;FOLD PLACE 3
;FOLD PROPRIEDADES
Ponto_STR[Pallet_2,Prdt_32BarPacking,3].NumCaixas = 3
Ponto_STR[Pallet_2,Prdt_32BarPacking,3].PickOp = 2
Ponto_STR[Pallet_2,Prdt_32BarPacking,3].ConfGarraOp = 3
Ponto_STR[Pallet_2,Prdt_32BarPacking,3].FechaGarraOp = 0
Ponto_STR[Pallet_2,Prdt_32BarPacking,3].AbreGarraOp = 0
Ponto_STR[Pallet_2,Prdt_32BarPacking,3].SensoresCaixa = 12345
Ponto_STR[Pallet_2,Prdt_32BarPacking,3].TravaGarra = False
Ponto_STR[Pallet_2,Prdt_32BarPacking,3].SkipGoHome = False
Ponto_STR[Pallet_2,Prdt_32BarPacking,3].SkipSobeRelAtual = False
Ponto_STR[Pallet_2,Prdt_32BarPacking,3].XApp1Place=P2_32BarPacking_3_App1
Ponto_STR[Pallet_2,Prdt_32BarPacking,3].XApp2Place=P2_32BarPacking_3_App2
Ponto_STR[Pallet_2,Prdt_32BarPacking,3].XPlace=P2_32BarPacking_3_Place
;ENDFOLD
;FOLD OffsetPlace
Ponto_STR[Pallet_2,Prdt_32BarPacking,3].OffsetPlace.X=0
Ponto_STR[Pallet_2,Prdt_32BarPacking,3].OffsetPlace.Y=0
Ponto_STR[Pallet_2,Prdt_32BarPacking,3].OffsetPlace.Z=0
Ponto_STR[Pallet_2,Prdt_32BarPacking,3].OffsetPlace.A=0
Ponto_STR[Pallet_2,Prdt_32BarPacking,3].OffsetPlace.B=0
Ponto_STR[Pallet_2,Prdt_32BarPacking,3].OffsetPlace.C=0
;ENDFOLD
;ENDFOLD

;ENDFOLD
;ENDFOLD

;FOLD Pallet 2 - Produto 33BarPacking
;FOLD LAYER 1: PLACE 1 ate 2
;FOLD PLACE 1
;FOLD PROPRIEDADES
Ponto_STR[Pallet_2,Prdt_33BarPacking,1].NumCaixas = 3
Ponto_STR[Pallet_2,Prdt_33BarPacking,1].PickOp = 2
Ponto_STR[Pallet_2,Prdt_33BarPacking,1].ConfGarraOp = 2
Ponto_STR[Pallet_2,Prdt_33BarPacking,1].FechaGarraOp = 0
Ponto_STR[Pallet_2,Prdt_33BarPacking,1].AbreGarraOp = 0
Ponto_STR[Pallet_2,Prdt_33BarPacking,1].SensoresCaixa = 12345
Ponto_STR[Pallet_2,Prdt_33BarPacking,1].TravaGarra = False
Ponto_STR[Pallet_2,Prdt_33BarPacking,1].SkipGoHome = False
Ponto_STR[Pallet_2,Prdt_33BarPacking,1].SkipSobeRelAtual = False
Ponto_STR[Pallet_2,Prdt_33BarPacking,1].XApp1Place=P2_33BarPacking_1_App1
Ponto_STR[Pallet_2,Prdt_33BarPacking,1].XApp2Place=P2_33BarPacking_1_App2
Ponto_STR[Pallet_2,Prdt_33BarPacking,1].XPlace=P2_33BarPacking_1_Place
;ENDFOLD
;FOLD OffsetPlace
Ponto_STR[Pallet_2,Prdt_33BarPacking,1].OffsetPlace.X=0
Ponto_STR[Pallet_2,Prdt_33BarPacking,1].OffsetPlace.Y=0
Ponto_STR[Pallet_2,Prdt_33BarPacking,1].OffsetPlace.Z=0
Ponto_STR[Pallet_2,Prdt_33BarPacking,1].OffsetPlace.A=0
Ponto_STR[Pallet_2,Prdt_33BarPacking,1].OffsetPlace.B=0
Ponto_STR[Pallet_2,Prdt_33BarPacking,1].OffsetPlace.C=0
;ENDFOLD
;ENDFOLD

;FOLD PLACE 2
;FOLD PROPRIEDADES
Ponto_STR[Pallet_2,Prdt_33BarPacking,2].NumCaixas = 3
Ponto_STR[Pallet_2,Prdt_33BarPacking,2].PickOp = 2
Ponto_STR[Pallet_2,Prdt_33BarPacking,2].ConfGarraOp = 2
Ponto_STR[Pallet_2,Prdt_33BarPacking,2].FechaGarraOp = 0
Ponto_STR[Pallet_2,Prdt_33BarPacking,2].AbreGarraOp = 0
Ponto_STR[Pallet_2,Prdt_33BarPacking,2].SensoresCaixa = 12345
Ponto_STR[Pallet_2,Prdt_33BarPacking,2].TravaGarra = False
Ponto_STR[Pallet_2,Prdt_33BarPacking,2].SkipGoHome = False
Ponto_STR[Pallet_2,Prdt_33BarPacking,2].SkipSobeRelAtual = False
Ponto_STR[Pallet_2,Prdt_33BarPacking,2].XApp1Place=P2_33BarPacking_2_App1
Ponto_STR[Pallet_2,Prdt_33BarPacking,2].XApp2Place=P2_33BarPacking_2_App2
Ponto_STR[Pallet_2,Prdt_33BarPacking,2].XPlace=P2_33BarPacking_2_Place
;ENDFOLD
;FOLD OffsetPlace
Ponto_STR[Pallet_2,Prdt_33BarPacking,2].OffsetPlace.X=0
Ponto_STR[Pallet_2,Prdt_33BarPacking,2].OffsetPlace.Y=0
Ponto_STR[Pallet_2,Prdt_33BarPacking,2].OffsetPlace.Z=0
Ponto_STR[Pallet_2,Prdt_33BarPacking,2].OffsetPlace.A=0
Ponto_STR[Pallet_2,Prdt_33BarPacking,2].OffsetPlace.B=0
Ponto_STR[Pallet_2,Prdt_33BarPacking,2].OffsetPlace.C=0
;ENDFOLD
;ENDFOLD

;ENDFOLD
;ENDFOLD

;FOLD Pallet 2 - Produto 34BarPacking
;FOLD LAYER 1: PLACE 1 ate 2
;FOLD PLACE 1
;FOLD PROPRIEDADES
Ponto_STR[Pallet_2,Prdt_34BarPacking,1].NumCaixas = 1
Ponto_STR[Pallet_2,Prdt_34BarPacking,1].PickOp = 3
Ponto_STR[Pallet_2,Prdt_34BarPacking,1].ConfGarraOp = 3
Ponto_STR[Pallet_2,Prdt_34BarPacking,1].FechaGarraOp = 0
Ponto_STR[Pallet_2,Prdt_34BarPacking,1].AbreGarraOp = 0
Ponto_STR[Pallet_2,Prdt_34BarPacking,1].SensoresCaixa = 123
Ponto_STR[Pallet_2,Prdt_34BarPacking,1].TravaGarra = False
Ponto_STR[Pallet_2,Prdt_34BarPacking,1].SkipGoHome = False
Ponto_STR[Pallet_2,Prdt_34BarPacking,1].SkipSobeRelAtual = False
Ponto_STR[Pallet_2,Prdt_34BarPacking,1].XApp1Place=P2_34BarPacking_1_App1
Ponto_STR[Pallet_2,Prdt_34BarPacking,1].XApp2Place=P2_34BarPacking_1_App2
Ponto_STR[Pallet_2,Prdt_34BarPacking,1].XPlace=P2_34BarPacking_1_Place
;ENDFOLD
;FOLD OffsetPlace
Ponto_STR[Pallet_2,Prdt_34BarPacking,1].OffsetPlace.X=0
Ponto_STR[Pallet_2,Prdt_34BarPacking,1].OffsetPlace.Y=0
Ponto_STR[Pallet_2,Prdt_34BarPacking,1].OffsetPlace.Z=0
Ponto_STR[Pallet_2,Prdt_34BarPacking,1].OffsetPlace.A=0
Ponto_STR[Pallet_2,Prdt_34BarPacking,1].OffsetPlace.B=0
Ponto_STR[Pallet_2,Prdt_34BarPacking,1].OffsetPlace.C=0
;ENDFOLD
;ENDFOLD

;FOLD PLACE 2
;FOLD PROPRIEDADES
Ponto_STR[Pallet_2,Prdt_34BarPacking,2].NumCaixas = 1
Ponto_STR[Pallet_2,Prdt_34BarPacking,2].PickOp = 3
Ponto_STR[Pallet_2,Prdt_34BarPacking,2].ConfGarraOp = 3
Ponto_STR[Pallet_2,Prdt_34BarPacking,2].FechaGarraOp = 0
Ponto_STR[Pallet_2,Prdt_34BarPacking,2].AbreGarraOp = 0
Ponto_STR[Pallet_2,Prdt_34BarPacking,2].SensoresCaixa = 123
Ponto_STR[Pallet_2,Prdt_34BarPacking,2].TravaGarra = False
Ponto_STR[Pallet_2,Prdt_34BarPacking,2].SkipGoHome = False
Ponto_STR[Pallet_2,Prdt_34BarPacking,2].SkipSobeRelAtual = False
Ponto_STR[Pallet_2,Prdt_34BarPacking,2].XApp1Place=P2_34BarPacking_2_App1
Ponto_STR[Pallet_2,Prdt_34BarPacking,2].XApp2Place=P2_34BarPacking_2_App2
Ponto_STR[Pallet_2,Prdt_34BarPacking,2].XPlace=P2_34BarPacking_2_Place
;ENDFOLD
;FOLD OffsetPlace
Ponto_STR[Pallet_2,Prdt_34BarPacking,2].OffsetPlace.X=0
Ponto_STR[Pallet_2,Prdt_34BarPacking,2].OffsetPlace.Y=0
Ponto_STR[Pallet_2,Prdt_34BarPacking,2].OffsetPlace.Z=0
Ponto_STR[Pallet_2,Prdt_34BarPacking,2].OffsetPlace.A=0
Ponto_STR[Pallet_2,Prdt_34BarPacking,2].OffsetPlace.B=0
Ponto_STR[Pallet_2,Prdt_34BarPacking,2].OffsetPlace.C=0
;ENDFOLD
;ENDFOLD

;ENDFOLD
;ENDFOLD

;FOLD Pallet 2 - Produto 9Aero
;FOLD LAYER 1: PLACE 1 ate 2
;FOLD PLACE 1
;FOLD PROPRIEDADES
Ponto_STR[Pallet_2,Prdt_9Aero,1].NumCaixas = 4
Ponto_STR[Pallet_2,Prdt_9Aero,1].PickOp = 3
Ponto_STR[Pallet_2,Prdt_9Aero,1].ConfGarraOp = 3
Ponto_STR[Pallet_2,Prdt_9Aero,1].FechaGarraOp = 0
Ponto_STR[Pallet_2,Prdt_9Aero,1].AbreGarraOp = 0
Ponto_STR[Pallet_2,Prdt_9Aero,1].SensoresCaixa = 123456
Ponto_STR[Pallet_2,Prdt_9Aero,1].TravaGarra = False
Ponto_STR[Pallet_2,Prdt_9Aero,1].SkipGoHome = False
Ponto_STR[Pallet_2,Prdt_9Aero,1].SkipSobeRelAtual = False
Ponto_STR[Pallet_2,Prdt_9Aero,1].XApp1Place=P2_9Aero_1_App1
Ponto_STR[Pallet_2,Prdt_9Aero,1].XApp2Place=P2_9Aero_1_App2
Ponto_STR[Pallet_2,Prdt_9Aero,1].XPlace=P2_9Aero_1_Place
;ENDFOLD
;FOLD OffsetPlace
Ponto_STR[Pallet_2,Prdt_9Aero,1].OffsetPlace.X=0
Ponto_STR[Pallet_2,Prdt_9Aero,1].OffsetPlace.Y=0
Ponto_STR[Pallet_2,Prdt_9Aero,1].OffsetPlace.Z=0
Ponto_STR[Pallet_2,Prdt_9Aero,1].OffsetPlace.A=0
Ponto_STR[Pallet_2,Prdt_9Aero,1].OffsetPlace.B=0
Ponto_STR[Pallet_2,Prdt_9Aero,1].OffsetPlace.C=0
;ENDFOLD
;ENDFOLD

;FOLD PLACE 2
;FOLD PROPRIEDADES
Ponto_STR[Pallet_2,Prdt_9Aero,2].NumCaixas = 4
Ponto_STR[Pallet_2,Prdt_9Aero,2].PickOp = 3
Ponto_STR[Pallet_2,Prdt_9Aero,2].ConfGarraOp = 3
Ponto_STR[Pallet_2,Prdt_9Aero,2].FechaGarraOp = 0
Ponto_STR[Pallet_2,Prdt_9Aero,2].AbreGarraOp = 0
Ponto_STR[Pallet_2,Prdt_9Aero,2].SensoresCaixa = 123456
Ponto_STR[Pallet_2,Prdt_9Aero,2].TravaGarra = False
Ponto_STR[Pallet_2,Prdt_9Aero,2].SkipGoHome = False
Ponto_STR[Pallet_2,Prdt_9Aero,2].SkipSobeRelAtual = False
Ponto_STR[Pallet_2,Prdt_9Aero,2].XApp1Place=P2_9Aero_2_App1
Ponto_STR[Pallet_2,Prdt_9Aero,2].XApp2Place=P2_9Aero_2_App2
Ponto_STR[Pallet_2,Prdt_9Aero,2].XPlace=P2_9Aero_2_Place
;ENDFOLD
;FOLD OffsetPlace
Ponto_STR[Pallet_2,Prdt_9Aero,2].OffsetPlace.X=0
Ponto_STR[Pallet_2,Prdt_9Aero,2].OffsetPlace.Y=0
Ponto_STR[Pallet_2,Prdt_9Aero,2].OffsetPlace.Z=0
Ponto_STR[Pallet_2,Prdt_9Aero,2].OffsetPlace.A=0
Ponto_STR[Pallet_2,Prdt_9Aero,2].OffsetPlace.B=0
Ponto_STR[Pallet_2,Prdt_9Aero,2].OffsetPlace.C=0
;ENDFOLD
;ENDFOLD

;ENDFOLD
;ENDFOLD

;FOLD Pallet 2 - Produto 23Smarties
;FOLD LAYER 1: PLACE 1 ate 4
;FOLD PLACE 1
;FOLD PROPRIEDADES
Ponto_STR[Pallet_2,Prdt_23Smarties,1].NumCaixas = 2
Ponto_STR[Pallet_2,Prdt_23Smarties,1].PickOp = 4
Ponto_STR[Pallet_2,Prdt_23Smarties,1].ConfGarraOp = 4
Ponto_STR[Pallet_2,Prdt_23Smarties,1].FechaGarraOp = 0
Ponto_STR[Pallet_2,Prdt_23Smarties,1].AbreGarraOp = 0
Ponto_STR[Pallet_2,Prdt_23Smarties,1].SensoresCaixa = 456
Ponto_STR[Pallet_2,Prdt_23Smarties,1].TravaGarra = False
Ponto_STR[Pallet_2,Prdt_23Smarties,1].SkipGoHome = False
Ponto_STR[Pallet_2,Prdt_23Smarties,1].SkipSobeRelAtual = False
Ponto_STR[Pallet_2,Prdt_23Smarties,1].XApp1Place=P2_23Smarties_1_App1
Ponto_STR[Pallet_2,Prdt_23Smarties,1].XApp2Place=P2_23Smarties_1_App2
Ponto_STR[Pallet_2,Prdt_23Smarties,1].XPlace=P2_23Smarties_1_Place
;ENDFOLD
;FOLD OffsetPlace
Ponto_STR[Pallet_2,Prdt_23Smarties,1].OffsetPlace.X=0
Ponto_STR[Pallet_2,Prdt_23Smarties,1].OffsetPlace.Y=0
Ponto_STR[Pallet_2,Prdt_23Smarties,1].OffsetPlace.Z=0
Ponto_STR[Pallet_2,Prdt_23Smarties,1].OffsetPlace.A=0
Ponto_STR[Pallet_2,Prdt_23Smarties,1].OffsetPlace.B=0
Ponto_STR[Pallet_2,Prdt_23Smarties,1].OffsetPlace.C=0
;ENDFOLD
;ENDFOLD

;FOLD PLACE 2
;FOLD PROPRIEDADES
Ponto_STR[Pallet_2,Prdt_23Smarties,2].NumCaixas = 3
Ponto_STR[Pallet_2,Prdt_23Smarties,2].PickOp = 4
Ponto_STR[Pallet_2,Prdt_23Smarties,2].ConfGarraOp = 4
Ponto_STR[Pallet_2,Prdt_23Smarties,2].FechaGarraOp = 0
Ponto_STR[Pallet_2,Prdt_23Smarties,2].AbreGarraOp = 0
Ponto_STR[Pallet_2,Prdt_23Smarties,2].SensoresCaixa = 3456
Ponto_STR[Pallet_2,Prdt_23Smarties,2].TravaGarra = False
Ponto_STR[Pallet_2,Prdt_23Smarties,2].SkipGoHome = False
Ponto_STR[Pallet_2,Prdt_23Smarties,2].SkipSobeRelAtual = False
Ponto_STR[Pallet_2,Prdt_23Smarties,2].XApp1Place=P2_23Smarties_2_App1
Ponto_STR[Pallet_2,Prdt_23Smarties,2].XApp2Place=P2_23Smarties_2_App2
Ponto_STR[Pallet_2,Prdt_23Smarties,2].XPlace=P2_23Smarties_2_Place
;ENDFOLD
;FOLD OffsetPlace
Ponto_STR[Pallet_2,Prdt_23Smarties,2].OffsetPlace.X=0
Ponto_STR[Pallet_2,Prdt_23Smarties,2].OffsetPlace.Y=0
Ponto_STR[Pallet_2,Prdt_23Smarties,2].OffsetPlace.Z=0
Ponto_STR[Pallet_2,Prdt_23Smarties,2].OffsetPlace.A=0
Ponto_STR[Pallet_2,Prdt_23Smarties,2].OffsetPlace.B=0
Ponto_STR[Pallet_2,Prdt_23Smarties,2].OffsetPlace.C=0
;ENDFOLD
;ENDFOLD

;FOLD PLACE 3
;FOLD PROPRIEDADES
Ponto_STR[Pallet_2,Prdt_23Smarties,3].NumCaixas = 2
Ponto_STR[Pallet_2,Prdt_23Smarties,3].PickOp = 4
Ponto_STR[Pallet_2,Prdt_23Smarties,3].ConfGarraOp = 4
Ponto_STR[Pallet_2,Prdt_23Smarties,3].FechaGarraOp = 0
Ponto_STR[Pallet_2,Prdt_23Smarties,3].AbreGarraOp = 0
Ponto_STR[Pallet_2,Prdt_23Smarties,3].SensoresCaixa = 456
Ponto_STR[Pallet_2,Prdt_23Smarties,3].TravaGarra = False
Ponto_STR[Pallet_2,Prdt_23Smarties,3].SkipGoHome = False
Ponto_STR[Pallet_2,Prdt_23Smarties,3].SkipSobeRelAtual = False
Ponto_STR[Pallet_2,Prdt_23Smarties,3].XApp1Place=P2_23Smarties_3_App1
Ponto_STR[Pallet_2,Prdt_23Smarties,3].XApp2Place=P2_23Smarties_3_App2
Ponto_STR[Pallet_2,Prdt_23Smarties,3].XPlace=P2_23Smarties_3_Place
;ENDFOLD
;FOLD OffsetPlace
Ponto_STR[Pallet_2,Prdt_23Smarties,3].OffsetPlace.X=0
Ponto_STR[Pallet_2,Prdt_23Smarties,3].OffsetPlace.Y=0
Ponto_STR[Pallet_2,Prdt_23Smarties,3].OffsetPlace.Z=0
Ponto_STR[Pallet_2,Prdt_23Smarties,3].OffsetPlace.A=0
Ponto_STR[Pallet_2,Prdt_23Smarties,3].OffsetPlace.B=0
Ponto_STR[Pallet_2,Prdt_23Smarties,3].OffsetPlace.C=0
;ENDFOLD
;ENDFOLD

;FOLD PLACE 4
;FOLD PROPRIEDADES
Ponto_STR[Pallet_2,Prdt_23Smarties,4].NumCaixas = 3
Ponto_STR[Pallet_2,Prdt_23Smarties,4].PickOp = 4
Ponto_STR[Pallet_2,Prdt_23Smarties,4].ConfGarraOp = 4
Ponto_STR[Pallet_2,Prdt_23Smarties,4].FechaGarraOp = 0
Ponto_STR[Pallet_2,Prdt_23Smarties,4].AbreGarraOp = 0
Ponto_STR[Pallet_2,Prdt_23Smarties,4].SensoresCaixa = 3456
Ponto_STR[Pallet_2,Prdt_23Smarties,4].TravaGarra = False
Ponto_STR[Pallet_2,Prdt_23Smarties,4].SkipGoHome = False
Ponto_STR[Pallet_2,Prdt_23Smarties,4].SkipSobeRelAtual = False
Ponto_STR[Pallet_2,Prdt_23Smarties,4].XApp1Place=P2_23Smarties_4_App1
Ponto_STR[Pallet_2,Prdt_23Smarties,4].XApp2Place=P2_23Smarties_4_App2
Ponto_STR[Pallet_2,Prdt_23Smarties,4].XPlace=P2_23Smarties_4_Place
;ENDFOLD
;FOLD OffsetPlace
Ponto_STR[Pallet_2,Prdt_23Smarties,4].OffsetPlace.X=0
Ponto_STR[Pallet_2,Prdt_23Smarties,4].OffsetPlace.Y=0
Ponto_STR[Pallet_2,Prdt_23Smarties,4].OffsetPlace.Z=0
Ponto_STR[Pallet_2,Prdt_23Smarties,4].OffsetPlace.A=0
Ponto_STR[Pallet_2,Prdt_23Smarties,4].OffsetPlace.B=0
Ponto_STR[Pallet_2,Prdt_23Smarties,4].OffsetPlace.C=0
;ENDFOLD
;ENDFOLD

;ENDFOLD
;FOLD LAYER 2: PLACE 5 ate 8
;FOLD PLACE 5
;FOLD PROPRIEDADES
Ponto_STR[Pallet_2,Prdt_23Smarties,5].NumCaixas = 2
Ponto_STR[Pallet_2,Prdt_23Smarties,5].PickOp = 5
Ponto_STR[Pallet_2,Prdt_23Smarties,5].ConfGarraOp = 4
Ponto_STR[Pallet_2,Prdt_23Smarties,5].FechaGarraOp = 0
Ponto_STR[Pallet_2,Prdt_23Smarties,5].AbreGarraOp = 0
Ponto_STR[Pallet_2,Prdt_23Smarties,5].SensoresCaixa = 123
Ponto_STR[Pallet_2,Prdt_23Smarties,5].TravaGarra = False
Ponto_STR[Pallet_2,Prdt_23Smarties,5].SkipGoHome = False
Ponto_STR[Pallet_2,Prdt_23Smarties,5].SkipSobeRelAtual = False
Ponto_STR[Pallet_2,Prdt_23Smarties,5].XApp1Place=P2_23Smarties_5_App1
Ponto_STR[Pallet_2,Prdt_23Smarties,5].XApp2Place=P2_23Smarties_5_App2
Ponto_STR[Pallet_2,Prdt_23Smarties,5].XPlace=P2_23Smarties_5_Place
;ENDFOLD
;FOLD OffsetPlace
Ponto_STR[Pallet_2,Prdt_23Smarties,5].OffsetPlace.X=0
Ponto_STR[Pallet_2,Prdt_23Smarties,5].OffsetPlace.Y=0
Ponto_STR[Pallet_2,Prdt_23Smarties,5].OffsetPlace.Z=0
Ponto_STR[Pallet_2,Prdt_23Smarties,5].OffsetPlace.A=0
Ponto_STR[Pallet_2,Prdt_23Smarties,5].OffsetPlace.B=0
Ponto_STR[Pallet_2,Prdt_23Smarties,5].OffsetPlace.C=0
;ENDFOLD
;ENDFOLD

;FOLD PLACE 6
;FOLD PROPRIEDADES
Ponto_STR[Pallet_2,Prdt_23Smarties,6].NumCaixas = 3
Ponto_STR[Pallet_2,Prdt_23Smarties,6].PickOp = 5
Ponto_STR[Pallet_2,Prdt_23Smarties,6].ConfGarraOp = 4
Ponto_STR[Pallet_2,Prdt_23Smarties,6].FechaGarraOp = 0
Ponto_STR[Pallet_2,Prdt_23Smarties,6].AbreGarraOp = 0
Ponto_STR[Pallet_2,Prdt_23Smarties,6].SensoresCaixa = 1234
Ponto_STR[Pallet_2,Prdt_23Smarties,6].TravaGarra = False
Ponto_STR[Pallet_2,Prdt_23Smarties,6].SkipGoHome = False
Ponto_STR[Pallet_2,Prdt_23Smarties,6].SkipSobeRelAtual = False
Ponto_STR[Pallet_2,Prdt_23Smarties,6].XApp1Place=P2_23Smarties_6_App1
Ponto_STR[Pallet_2,Prdt_23Smarties,6].XApp2Place=P2_23Smarties_6_App2
Ponto_STR[Pallet_2,Prdt_23Smarties,6].XPlace=P2_23Smarties_6_Place
;ENDFOLD
;FOLD OffsetPlace
Ponto_STR[Pallet_2,Prdt_23Smarties,6].OffsetPlace.X=0
Ponto_STR[Pallet_2,Prdt_23Smarties,6].OffsetPlace.Y=0
Ponto_STR[Pallet_2,Prdt_23Smarties,6].OffsetPlace.Z=0
Ponto_STR[Pallet_2,Prdt_23Smarties,6].OffsetPlace.A=0
Ponto_STR[Pallet_2,Prdt_23Smarties,6].OffsetPlace.B=0
Ponto_STR[Pallet_2,Prdt_23Smarties,6].OffsetPlace.C=0
;ENDFOLD
;ENDFOLD

;FOLD PLACE 7
;FOLD PROPRIEDADES
Ponto_STR[Pallet_2,Prdt_23Smarties,7].NumCaixas = 2
Ponto_STR[Pallet_2,Prdt_23Smarties,7].PickOp = 5
Ponto_STR[Pallet_2,Prdt_23Smarties,7].ConfGarraOp = 4
Ponto_STR[Pallet_2,Prdt_23Smarties,7].FechaGarraOp = 0
Ponto_STR[Pallet_2,Prdt_23Smarties,7].AbreGarraOp = 0
Ponto_STR[Pallet_2,Prdt_23Smarties,7].SensoresCaixa = 123
Ponto_STR[Pallet_2,Prdt_23Smarties,7].TravaGarra = False
Ponto_STR[Pallet_2,Prdt_23Smarties,7].SkipGoHome = False
Ponto_STR[Pallet_2,Prdt_23Smarties,7].SkipSobeRelAtual = False
Ponto_STR[Pallet_2,Prdt_23Smarties,7].XApp1Place=P2_23Smarties_7_App1
Ponto_STR[Pallet_2,Prdt_23Smarties,7].XApp2Place=P2_23Smarties_7_App2
Ponto_STR[Pallet_2,Prdt_23Smarties,7].XPlace=P2_23Smarties_7_Place
;ENDFOLD
;FOLD OffsetPlace
Ponto_STR[Pallet_2,Prdt_23Smarties,7].OffsetPlace.X=0
Ponto_STR[Pallet_2,Prdt_23Smarties,7].OffsetPlace.Y=0
Ponto_STR[Pallet_2,Prdt_23Smarties,7].OffsetPlace.Z=0
Ponto_STR[Pallet_2,Prdt_23Smarties,7].OffsetPlace.A=0
Ponto_STR[Pallet_2,Prdt_23Smarties,7].OffsetPlace.B=0
Ponto_STR[Pallet_2,Prdt_23Smarties,7].OffsetPlace.C=0
;ENDFOLD
;ENDFOLD

;FOLD PLACE 8
;FOLD PROPRIEDADES
Ponto_STR[Pallet_2,Prdt_23Smarties,8].NumCaixas = 3
Ponto_STR[Pallet_2,Prdt_23Smarties,8].PickOp = 5
Ponto_STR[Pallet_2,Prdt_23Smarties,8].ConfGarraOp = 4
Ponto_STR[Pallet_2,Prdt_23Smarties,8].FechaGarraOp = 0
Ponto_STR[Pallet_2,Prdt_23Smarties,8].AbreGarraOp = 0
Ponto_STR[Pallet_2,Prdt_23Smarties,8].SensoresCaixa = 1234
Ponto_STR[Pallet_2,Prdt_23Smarties,8].TravaGarra = False
Ponto_STR[Pallet_2,Prdt_23Smarties,8].SkipGoHome = False
Ponto_STR[Pallet_2,Prdt_23Smarties,8].SkipSobeRelAtual = False
Ponto_STR[Pallet_2,Prdt_23Smarties,8].XApp1Place=P2_23Smarties_8_App1
Ponto_STR[Pallet_2,Prdt_23Smarties,8].XApp2Place=P2_23Smarties_8_App2
Ponto_STR[Pallet_2,Prdt_23Smarties,8].XPlace=P2_23Smarties_8_Place
;ENDFOLD
;FOLD OffsetPlace
Ponto_STR[Pallet_2,Prdt_23Smarties,8].OffsetPlace.X=0
Ponto_STR[Pallet_2,Prdt_23Smarties,8].OffsetPlace.Y=0
Ponto_STR[Pallet_2,Prdt_23Smarties,8].OffsetPlace.Z=0
Ponto_STR[Pallet_2,Prdt_23Smarties,8].OffsetPlace.A=0
Ponto_STR[Pallet_2,Prdt_23Smarties,8].OffsetPlace.B=0
Ponto_STR[Pallet_2,Prdt_23Smarties,8].OffsetPlace.C=0
;ENDFOLD
;ENDFOLD

;ENDFOLD
;ENDFOLD

;FOLD Pallet 2 - Produto 10CoffeCrisp
;FOLD LAYER 1: PLACE 1 ate 4
;FOLD PLACE 1
;FOLD PROPRIEDADES
Ponto_STR[Pallet_2,Prdt_10CoffeCrisp,1].NumCaixas = 1
Ponto_STR[Pallet_2,Prdt_10CoffeCrisp,1].PickOp = 6
Ponto_STR[Pallet_2,Prdt_10CoffeCrisp,1].ConfGarraOp = 0
Ponto_STR[Pallet_2,Prdt_10CoffeCrisp,1].FechaGarraOp = 0
Ponto_STR[Pallet_2,Prdt_10CoffeCrisp,1].AbreGarraOp = 0
Ponto_STR[Pallet_2,Prdt_10CoffeCrisp,1].SensoresCaixa = 56
Ponto_STR[Pallet_2,Prdt_10CoffeCrisp,1].TravaGarra = False
Ponto_STR[Pallet_2,Prdt_10CoffeCrisp,1].SkipGoHome = False
Ponto_STR[Pallet_2,Prdt_10CoffeCrisp,1].SkipSobeRelAtual = False
Ponto_STR[Pallet_2,Prdt_10CoffeCrisp,1].XApp1Place=P2_10CoffeCrisp_1_App1
Ponto_STR[Pallet_2,Prdt_10CoffeCrisp,1].XApp2Place=P2_10CoffeCrisp_1_App2
Ponto_STR[Pallet_2,Prdt_10CoffeCrisp,1].XPlace=P2_10CoffeCrisp_1_Place
;ENDFOLD
;FOLD OffsetPlace
Ponto_STR[Pallet_2,Prdt_10CoffeCrisp,1].OffsetPlace.X=0
Ponto_STR[Pallet_2,Prdt_10CoffeCrisp,1].OffsetPlace.Y=0
Ponto_STR[Pallet_2,Prdt_10CoffeCrisp,1].OffsetPlace.Z=0
Ponto_STR[Pallet_2,Prdt_10CoffeCrisp,1].OffsetPlace.A=0
Ponto_STR[Pallet_2,Prdt_10CoffeCrisp,1].OffsetPlace.B=0
Ponto_STR[Pallet_2,Prdt_10CoffeCrisp,1].OffsetPlace.C=0
;ENDFOLD
;ENDFOLD

;FOLD PLACE 2
;FOLD PROPRIEDADES
Ponto_STR[Pallet_2,Prdt_10CoffeCrisp,2].NumCaixas = 1
Ponto_STR[Pallet_2,Prdt_10CoffeCrisp,2].PickOp = 6
Ponto_STR[Pallet_2,Prdt_10CoffeCrisp,2].ConfGarraOp = 0
Ponto_STR[Pallet_2,Prdt_10CoffeCrisp,2].FechaGarraOp = 0
Ponto_STR[Pallet_2,Prdt_10CoffeCrisp,2].AbreGarraOp = 0
Ponto_STR[Pallet_2,Prdt_10CoffeCrisp,2].SensoresCaixa = 56
Ponto_STR[Pallet_2,Prdt_10CoffeCrisp,2].TravaGarra = False
Ponto_STR[Pallet_2,Prdt_10CoffeCrisp,2].SkipGoHome = False
Ponto_STR[Pallet_2,Prdt_10CoffeCrisp,2].SkipSobeRelAtual = False
Ponto_STR[Pallet_2,Prdt_10CoffeCrisp,2].XApp1Place=P2_10CoffeCrisp_2_App1
Ponto_STR[Pallet_2,Prdt_10CoffeCrisp,2].XApp2Place=P2_10CoffeCrisp_2_App2
Ponto_STR[Pallet_2,Prdt_10CoffeCrisp,2].XPlace=P2_10CoffeCrisp_2_Place
;ENDFOLD
;FOLD OffsetPlace
Ponto_STR[Pallet_2,Prdt_10CoffeCrisp,2].OffsetPlace.X=0
Ponto_STR[Pallet_2,Prdt_10CoffeCrisp,2].OffsetPlace.Y=0
Ponto_STR[Pallet_2,Prdt_10CoffeCrisp,2].OffsetPlace.Z=0
Ponto_STR[Pallet_2,Prdt_10CoffeCrisp,2].OffsetPlace.A=0
Ponto_STR[Pallet_2,Prdt_10CoffeCrisp,2].OffsetPlace.B=0
Ponto_STR[Pallet_2,Prdt_10CoffeCrisp,2].OffsetPlace.C=0
;ENDFOLD
;ENDFOLD

;FOLD PLACE 3
;FOLD PROPRIEDADES
Ponto_STR[Pallet_2,Prdt_10CoffeCrisp,3].NumCaixas = 3
Ponto_STR[Pallet_2,Prdt_10CoffeCrisp,3].PickOp = 1
Ponto_STR[Pallet_2,Prdt_10CoffeCrisp,3].ConfGarraOp = 0
Ponto_STR[Pallet_2,Prdt_10CoffeCrisp,3].FechaGarraOp = 0
Ponto_STR[Pallet_2,Prdt_10CoffeCrisp,3].AbreGarraOp = 0
Ponto_STR[Pallet_2,Prdt_10CoffeCrisp,3].SensoresCaixa = 12345
Ponto_STR[Pallet_2,Prdt_10CoffeCrisp,3].TravaGarra = False
Ponto_STR[Pallet_2,Prdt_10CoffeCrisp,3].SkipGoHome = False
Ponto_STR[Pallet_2,Prdt_10CoffeCrisp,3].SkipSobeRelAtual = False
Ponto_STR[Pallet_2,Prdt_10CoffeCrisp,3].XApp1Place=P2_10CoffeCrisp_3_App1
Ponto_STR[Pallet_2,Prdt_10CoffeCrisp,3].XApp2Place=P2_10CoffeCrisp_3_App2
Ponto_STR[Pallet_2,Prdt_10CoffeCrisp,3].XPlace=P2_10CoffeCrisp_3_Place
;ENDFOLD
;FOLD OffsetPlace
Ponto_STR[Pallet_2,Prdt_10CoffeCrisp,3].OffsetPlace.X=0
Ponto_STR[Pallet_2,Prdt_10CoffeCrisp,3].OffsetPlace.Y=0
Ponto_STR[Pallet_2,Prdt_10CoffeCrisp,3].OffsetPlace.Z=0
Ponto_STR[Pallet_2,Prdt_10CoffeCrisp,3].OffsetPlace.A=0
Ponto_STR[Pallet_2,Prdt_10CoffeCrisp,3].OffsetPlace.B=0
Ponto_STR[Pallet_2,Prdt_10CoffeCrisp,3].OffsetPlace.C=0
;ENDFOLD
;ENDFOLD

;FOLD PLACE 4
;FOLD PROPRIEDADES
Ponto_STR[Pallet_2,Prdt_10CoffeCrisp,4].NumCaixas = 3
Ponto_STR[Pallet_2,Prdt_10CoffeCrisp,4].PickOp = 1
Ponto_STR[Pallet_2,Prdt_10CoffeCrisp,4].ConfGarraOp = 0
Ponto_STR[Pallet_2,Prdt_10CoffeCrisp,4].FechaGarraOp = 0
Ponto_STR[Pallet_2,Prdt_10CoffeCrisp,4].AbreGarraOp = 0
Ponto_STR[Pallet_2,Prdt_10CoffeCrisp,4].SensoresCaixa = 12345
Ponto_STR[Pallet_2,Prdt_10CoffeCrisp,4].TravaGarra = False
Ponto_STR[Pallet_2,Prdt_10CoffeCrisp,4].SkipGoHome = False
Ponto_STR[Pallet_2,Prdt_10CoffeCrisp,4].SkipSobeRelAtual = False
Ponto_STR[Pallet_2,Prdt_10CoffeCrisp,4].XApp1Place=P2_10CoffeCrisp_4_App1
Ponto_STR[Pallet_2,Prdt_10CoffeCrisp,4].XApp2Place=P2_10CoffeCrisp_4_App2
Ponto_STR[Pallet_2,Prdt_10CoffeCrisp,4].XPlace=P2_10CoffeCrisp_4_Place
;ENDFOLD
;FOLD OffsetPlace
Ponto_STR[Pallet_2,Prdt_10CoffeCrisp,4].OffsetPlace.X=0
Ponto_STR[Pallet_2,Prdt_10CoffeCrisp,4].OffsetPlace.Y=0
Ponto_STR[Pallet_2,Prdt_10CoffeCrisp,4].OffsetPlace.Z=0
Ponto_STR[Pallet_2,Prdt_10CoffeCrisp,4].OffsetPlace.A=0
Ponto_STR[Pallet_2,Prdt_10CoffeCrisp,4].OffsetPlace.B=0
Ponto_STR[Pallet_2,Prdt_10CoffeCrisp,4].OffsetPlace.C=0
;ENDFOLD
;ENDFOLD

;ENDFOLD
;FOLD LAYER 2: PLACE 5 ate 8
;FOLD PLACE 5
;FOLD PROPRIEDADES
Ponto_STR[Pallet_2,Prdt_10CoffeCrisp,5].NumCaixas = 1
Ponto_STR[Pallet_2,Prdt_10CoffeCrisp,5].PickOp = 3
Ponto_STR[Pallet_2,Prdt_10CoffeCrisp,5].ConfGarraOp = 3
Ponto_STR[Pallet_2,Prdt_10CoffeCrisp,5].FechaGarraOp = 0
Ponto_STR[Pallet_2,Prdt_10CoffeCrisp,5].AbreGarraOp = 0
Ponto_STR[Pallet_2,Prdt_10CoffeCrisp,5].SensoresCaixa = 12
Ponto_STR[Pallet_2,Prdt_10CoffeCrisp,5].TravaGarra = False
Ponto_STR[Pallet_2,Prdt_10CoffeCrisp,5].SkipGoHome = False
Ponto_STR[Pallet_2,Prdt_10CoffeCrisp,5].SkipSobeRelAtual = False
Ponto_STR[Pallet_2,Prdt_10CoffeCrisp,5].XApp1Place=P2_10CoffeCrisp_5_App1
Ponto_STR[Pallet_2,Prdt_10CoffeCrisp,5].XApp2Place=P2_10CoffeCrisp_5_App2
Ponto_STR[Pallet_2,Prdt_10CoffeCrisp,5].XPlace=P2_10CoffeCrisp_5_Place
;ENDFOLD
;FOLD OffsetPlace
Ponto_STR[Pallet_2,Prdt_10CoffeCrisp,5].OffsetPlace.X=0
Ponto_STR[Pallet_2,Prdt_10CoffeCrisp,5].OffsetPlace.Y=0
Ponto_STR[Pallet_2,Prdt_10CoffeCrisp,5].OffsetPlace.Z=0
Ponto_STR[Pallet_2,Prdt_10CoffeCrisp,5].OffsetPlace.A=0
Ponto_STR[Pallet_2,Prdt_10CoffeCrisp,5].OffsetPlace.B=0
Ponto_STR[Pallet_2,Prdt_10CoffeCrisp,5].OffsetPlace.C=0
;ENDFOLD
;ENDFOLD

;FOLD PLACE 6
;FOLD PROPRIEDADES
Ponto_STR[Pallet_2,Prdt_10CoffeCrisp,6].NumCaixas = 1
Ponto_STR[Pallet_2,Prdt_10CoffeCrisp,6].PickOp = 3
Ponto_STR[Pallet_2,Prdt_10CoffeCrisp,6].ConfGarraOp = 3
Ponto_STR[Pallet_2,Prdt_10CoffeCrisp,6].FechaGarraOp = 0
Ponto_STR[Pallet_2,Prdt_10CoffeCrisp,6].AbreGarraOp = 0
Ponto_STR[Pallet_2,Prdt_10CoffeCrisp,6].SensoresCaixa = 12
Ponto_STR[Pallet_2,Prdt_10CoffeCrisp,6].TravaGarra = False
Ponto_STR[Pallet_2,Prdt_10CoffeCrisp,6].SkipGoHome = False
Ponto_STR[Pallet_2,Prdt_10CoffeCrisp,6].SkipSobeRelAtual = False
Ponto_STR[Pallet_2,Prdt_10CoffeCrisp,6].XApp1Place=P2_10CoffeCrisp_6_App1
Ponto_STR[Pallet_2,Prdt_10CoffeCrisp,6].XApp2Place=P2_10CoffeCrisp_6_App2
Ponto_STR[Pallet_2,Prdt_10CoffeCrisp,6].XPlace=P2_10CoffeCrisp_6_Place
;ENDFOLD
;FOLD OffsetPlace
Ponto_STR[Pallet_2,Prdt_10CoffeCrisp,6].OffsetPlace.X=0
Ponto_STR[Pallet_2,Prdt_10CoffeCrisp,6].OffsetPlace.Y=0
Ponto_STR[Pallet_2,Prdt_10CoffeCrisp,6].OffsetPlace.Z=0
Ponto_STR[Pallet_2,Prdt_10CoffeCrisp,6].OffsetPlace.A=0
Ponto_STR[Pallet_2,Prdt_10CoffeCrisp,6].OffsetPlace.B=0
Ponto_STR[Pallet_2,Prdt_10CoffeCrisp,6].OffsetPlace.C=0
;ENDFOLD
;ENDFOLD

;FOLD PLACE 7
;FOLD PROPRIEDADES
Ponto_STR[Pallet_2,Prdt_10CoffeCrisp,7].NumCaixas = 3
Ponto_STR[Pallet_2,Prdt_10CoffeCrisp,7].PickOp = 1
Ponto_STR[Pallet_2,Prdt_10CoffeCrisp,7].ConfGarraOp = 0
Ponto_STR[Pallet_2,Prdt_10CoffeCrisp,7].FechaGarraOp = 0
Ponto_STR[Pallet_2,Prdt_10CoffeCrisp,7].AbreGarraOp = 1
Ponto_STR[Pallet_2,Prdt_10CoffeCrisp,7].SensoresCaixa = 12345
Ponto_STR[Pallet_2,Prdt_10CoffeCrisp,7].TravaGarra = True
Ponto_STR[Pallet_2,Prdt_10CoffeCrisp,7].SkipGoHome = False
Ponto_STR[Pallet_2,Prdt_10CoffeCrisp,7].SkipSobeRelAtual = False
Ponto_STR[Pallet_2,Prdt_10CoffeCrisp,7].XApp1Place=P2_10CoffeCrisp_7_App1
Ponto_STR[Pallet_2,Prdt_10CoffeCrisp,7].XApp2Place=P2_10CoffeCrisp_7_App2
Ponto_STR[Pallet_2,Prdt_10CoffeCrisp,7].XPlace=P2_10CoffeCrisp_7_Place
;ENDFOLD
;FOLD OffsetPlace
Ponto_STR[Pallet_2,Prdt_10CoffeCrisp,7].OffsetPlace.X=0
Ponto_STR[Pallet_2,Prdt_10CoffeCrisp,7].OffsetPlace.Y=0
Ponto_STR[Pallet_2,Prdt_10CoffeCrisp,7].OffsetPlace.Z=0
Ponto_STR[Pallet_2,Prdt_10CoffeCrisp,7].OffsetPlace.A=0
Ponto_STR[Pallet_2,Prdt_10CoffeCrisp,7].OffsetPlace.B=0
Ponto_STR[Pallet_2,Prdt_10CoffeCrisp,7].OffsetPlace.C=0
;ENDFOLD
;ENDFOLD

;FOLD PLACE 8
;FOLD PROPRIEDADES
Ponto_STR[Pallet_2,Prdt_10CoffeCrisp,8].NumCaixas = 3
Ponto_STR[Pallet_2,Prdt_10CoffeCrisp,8].PickOp = 1
Ponto_STR[Pallet_2,Prdt_10CoffeCrisp,8].ConfGarraOp = 0
Ponto_STR[Pallet_2,Prdt_10CoffeCrisp,8].FechaGarraOp = 0
Ponto_STR[Pallet_2,Prdt_10CoffeCrisp,8].AbreGarraOp = 1
Ponto_STR[Pallet_2,Prdt_10CoffeCrisp,8].SensoresCaixa = 12345
Ponto_STR[Pallet_2,Prdt_10CoffeCrisp,8].TravaGarra = True
Ponto_STR[Pallet_2,Prdt_10CoffeCrisp,8].SkipGoHome = False
Ponto_STR[Pallet_2,Prdt_10CoffeCrisp,8].SkipSobeRelAtual = False
Ponto_STR[Pallet_2,Prdt_10CoffeCrisp,8].XApp1Place=P2_10CoffeCrisp_8_App1
Ponto_STR[Pallet_2,Prdt_10CoffeCrisp,8].XApp2Place=P2_10CoffeCrisp_8_App2
Ponto_STR[Pallet_2,Prdt_10CoffeCrisp,8].XPlace=P2_10CoffeCrisp_8_Place
;ENDFOLD
;FOLD OffsetPlace
Ponto_STR[Pallet_2,Prdt_10CoffeCrisp,8].OffsetPlace.X=0
Ponto_STR[Pallet_2,Prdt_10CoffeCrisp,8].OffsetPlace.Y=0
Ponto_STR[Pallet_2,Prdt_10CoffeCrisp,8].OffsetPlace.Z=0
Ponto_STR[Pallet_2,Prdt_10CoffeCrisp,8].OffsetPlace.A=0
Ponto_STR[Pallet_2,Prdt_10CoffeCrisp,8].OffsetPlace.B=0
Ponto_STR[Pallet_2,Prdt_10CoffeCrisp,8].OffsetPlace.C=0
;ENDFOLD
;ENDFOLD

;ENDFOLD
;ENDFOLD

;FOLD Pallet 2 - Produto 19KitKat
;FOLD LAYER 1: PLACE 1 ate 6
;FOLD PLACE 1
;FOLD PROPRIEDADES
Ponto_STR[Pallet_2,Prdt_19KitKat,1].NumCaixas = 1
Ponto_STR[Pallet_2,Prdt_19KitKat,1].PickOp = 6
Ponto_STR[Pallet_2,Prdt_19KitKat,1].ConfGarraOp = 0
Ponto_STR[Pallet_2,Prdt_19KitKat,1].FechaGarraOp = 0
Ponto_STR[Pallet_2,Prdt_19KitKat,1].AbreGarraOp = 0
Ponto_STR[Pallet_2,Prdt_19KitKat,1].SensoresCaixa = 6
Ponto_STR[Pallet_2,Prdt_19KitKat,1].TravaGarra = False
Ponto_STR[Pallet_2,Prdt_19KitKat,1].SkipGoHome = False
Ponto_STR[Pallet_2,Prdt_19KitKat,1].SkipSobeRelAtual = False
Ponto_STR[Pallet_2,Prdt_19KitKat,1].XApp1Place=P2_19KitKat_1_App1
Ponto_STR[Pallet_2,Prdt_19KitKat,1].XApp2Place=P2_19KitKat_1_App2
Ponto_STR[Pallet_2,Prdt_19KitKat,1].XPlace=P2_19KitKat_1_Place
;ENDFOLD
;FOLD OffsetPlace
Ponto_STR[Pallet_2,Prdt_19KitKat,1].OffsetPlace.X=0
Ponto_STR[Pallet_2,Prdt_19KitKat,1].OffsetPlace.Y=0
Ponto_STR[Pallet_2,Prdt_19KitKat,1].OffsetPlace.Z=0
Ponto_STR[Pallet_2,Prdt_19KitKat,1].OffsetPlace.A=0
Ponto_STR[Pallet_2,Prdt_19KitKat,1].OffsetPlace.B=0
Ponto_STR[Pallet_2,Prdt_19KitKat,1].OffsetPlace.C=0
;ENDFOLD
;ENDFOLD

;FOLD PLACE 2
;FOLD PROPRIEDADES
Ponto_STR[Pallet_2,Prdt_19KitKat,2].NumCaixas = 1
Ponto_STR[Pallet_2,Prdt_19KitKat,2].PickOp = 6
Ponto_STR[Pallet_2,Prdt_19KitKat,2].ConfGarraOp = 0
Ponto_STR[Pallet_2,Prdt_19KitKat,2].FechaGarraOp = 0
Ponto_STR[Pallet_2,Prdt_19KitKat,2].AbreGarraOp = 0
Ponto_STR[Pallet_2,Prdt_19KitKat,2].SensoresCaixa = 6
Ponto_STR[Pallet_2,Prdt_19KitKat,2].TravaGarra = False
Ponto_STR[Pallet_2,Prdt_19KitKat,2].SkipGoHome = False
Ponto_STR[Pallet_2,Prdt_19KitKat,2].SkipSobeRelAtual = False
Ponto_STR[Pallet_2,Prdt_19KitKat,2].XApp1Place=P2_19KitKat_2_App1
Ponto_STR[Pallet_2,Prdt_19KitKat,2].XApp2Place=P2_19KitKat_2_App2
Ponto_STR[Pallet_2,Prdt_19KitKat,2].XPlace=P2_19KitKat_2_Place
;ENDFOLD
;FOLD OffsetPlace
Ponto_STR[Pallet_2,Prdt_19KitKat,2].OffsetPlace.X=0
Ponto_STR[Pallet_2,Prdt_19KitKat,2].OffsetPlace.Y=0
Ponto_STR[Pallet_2,Prdt_19KitKat,2].OffsetPlace.Z=0
Ponto_STR[Pallet_2,Prdt_19KitKat,2].OffsetPlace.A=0
Ponto_STR[Pallet_2,Prdt_19KitKat,2].OffsetPlace.B=0
Ponto_STR[Pallet_2,Prdt_19KitKat,2].OffsetPlace.C=0
;ENDFOLD
;ENDFOLD

;FOLD PLACE 3
;FOLD PROPRIEDADES
Ponto_STR[Pallet_2,Prdt_19KitKat,3].NumCaixas = 1
Ponto_STR[Pallet_2,Prdt_19KitKat,3].PickOp = 6
Ponto_STR[Pallet_2,Prdt_19KitKat,3].ConfGarraOp = 0
Ponto_STR[Pallet_2,Prdt_19KitKat,3].FechaGarraOp = 0
Ponto_STR[Pallet_2,Prdt_19KitKat,3].AbreGarraOp = 0
Ponto_STR[Pallet_2,Prdt_19KitKat,3].SensoresCaixa = 6
Ponto_STR[Pallet_2,Prdt_19KitKat,3].TravaGarra = False
Ponto_STR[Pallet_2,Prdt_19KitKat,3].SkipGoHome = False
Ponto_STR[Pallet_2,Prdt_19KitKat,3].SkipSobeRelAtual = False
Ponto_STR[Pallet_2,Prdt_19KitKat,3].XApp1Place=P2_19KitKat_3_App1
Ponto_STR[Pallet_2,Prdt_19KitKat,3].XApp2Place=P2_19KitKat_3_App2
Ponto_STR[Pallet_2,Prdt_19KitKat,3].XPlace=P2_19KitKat_3_Place
;ENDFOLD
;FOLD OffsetPlace
Ponto_STR[Pallet_2,Prdt_19KitKat,3].OffsetPlace.X=0
Ponto_STR[Pallet_2,Prdt_19KitKat,3].OffsetPlace.Y=0
Ponto_STR[Pallet_2,Prdt_19KitKat,3].OffsetPlace.Z=0
Ponto_STR[Pallet_2,Prdt_19KitKat,3].OffsetPlace.A=0
Ponto_STR[Pallet_2,Prdt_19KitKat,3].OffsetPlace.B=0
Ponto_STR[Pallet_2,Prdt_19KitKat,3].OffsetPlace.C=0
;ENDFOLD
;ENDFOLD

;FOLD PLACE 4
;FOLD PROPRIEDADES
Ponto_STR[Pallet_2,Prdt_19KitKat,4].NumCaixas = 4
Ponto_STR[Pallet_2,Prdt_19KitKat,4].PickOp = 1
Ponto_STR[Pallet_2,Prdt_19KitKat,4].ConfGarraOp = 0
Ponto_STR[Pallet_2,Prdt_19KitKat,4].FechaGarraOp = 0
Ponto_STR[Pallet_2,Prdt_19KitKat,4].AbreGarraOp = 0
Ponto_STR[Pallet_2,Prdt_19KitKat,4].SensoresCaixa = 12345
Ponto_STR[Pallet_2,Prdt_19KitKat,4].TravaGarra = False
Ponto_STR[Pallet_2,Prdt_19KitKat,4].SkipGoHome = False
Ponto_STR[Pallet_2,Prdt_19KitKat,4].SkipSobeRelAtual = False
Ponto_STR[Pallet_2,Prdt_19KitKat,4].XApp1Place=P2_19KitKat_4_App1
Ponto_STR[Pallet_2,Prdt_19KitKat,4].XApp2Place=P2_19KitKat_4_App2
Ponto_STR[Pallet_2,Prdt_19KitKat,4].XPlace=P2_19KitKat_4_Place
;ENDFOLD
;FOLD OffsetPlace
Ponto_STR[Pallet_2,Prdt_19KitKat,4].OffsetPlace.X=0
Ponto_STR[Pallet_2,Prdt_19KitKat,4].OffsetPlace.Y=0
Ponto_STR[Pallet_2,Prdt_19KitKat,4].OffsetPlace.Z=0
Ponto_STR[Pallet_2,Prdt_19KitKat,4].OffsetPlace.A=0
Ponto_STR[Pallet_2,Prdt_19KitKat,4].OffsetPlace.B=0
Ponto_STR[Pallet_2,Prdt_19KitKat,4].OffsetPlace.C=0
;ENDFOLD
;ENDFOLD

;FOLD PLACE 5
;FOLD PROPRIEDADES
Ponto_STR[Pallet_2,Prdt_19KitKat,5].NumCaixas = 4
Ponto_STR[Pallet_2,Prdt_19KitKat,5].PickOp = 1
Ponto_STR[Pallet_2,Prdt_19KitKat,5].ConfGarraOp = 0
Ponto_STR[Pallet_2,Prdt_19KitKat,5].FechaGarraOp = 0
Ponto_STR[Pallet_2,Prdt_19KitKat,5].AbreGarraOp = 0
Ponto_STR[Pallet_2,Prdt_19KitKat,5].SensoresCaixa = 12345
Ponto_STR[Pallet_2,Prdt_19KitKat,5].TravaGarra = False
Ponto_STR[Pallet_2,Prdt_19KitKat,5].SkipGoHome = False
Ponto_STR[Pallet_2,Prdt_19KitKat,5].SkipSobeRelAtual = False
Ponto_STR[Pallet_2,Prdt_19KitKat,5].XApp1Place=P2_19KitKat_5_App1
Ponto_STR[Pallet_2,Prdt_19KitKat,5].XApp2Place=P2_19KitKat_5_App2
Ponto_STR[Pallet_2,Prdt_19KitKat,5].XPlace=P2_19KitKat_5_Place
;ENDFOLD
;FOLD OffsetPlace
Ponto_STR[Pallet_2,Prdt_19KitKat,5].OffsetPlace.X=0
Ponto_STR[Pallet_2,Prdt_19KitKat,5].OffsetPlace.Y=0
Ponto_STR[Pallet_2,Prdt_19KitKat,5].OffsetPlace.Z=0
Ponto_STR[Pallet_2,Prdt_19KitKat,5].OffsetPlace.A=0
Ponto_STR[Pallet_2,Prdt_19KitKat,5].OffsetPlace.B=0
Ponto_STR[Pallet_2,Prdt_19KitKat,5].OffsetPlace.C=0
;ENDFOLD
;ENDFOLD

;FOLD PLACE 6
;FOLD PROPRIEDADES
Ponto_STR[Pallet_2,Prdt_19KitKat,6].NumCaixas = 4
Ponto_STR[Pallet_2,Prdt_19KitKat,6].PickOp = 1
Ponto_STR[Pallet_2,Prdt_19KitKat,6].ConfGarraOp = 0
Ponto_STR[Pallet_2,Prdt_19KitKat,6].FechaGarraOp = 0
Ponto_STR[Pallet_2,Prdt_19KitKat,6].AbreGarraOp = 0
Ponto_STR[Pallet_2,Prdt_19KitKat,6].SensoresCaixa = 12345
Ponto_STR[Pallet_2,Prdt_19KitKat,6].TravaGarra = False
Ponto_STR[Pallet_2,Prdt_19KitKat,6].SkipGoHome = False
Ponto_STR[Pallet_2,Prdt_19KitKat,6].SkipSobeRelAtual = False
Ponto_STR[Pallet_2,Prdt_19KitKat,6].XApp1Place=P2_19KitKat_6_App1
Ponto_STR[Pallet_2,Prdt_19KitKat,6].XApp2Place=P2_19KitKat_6_App2
Ponto_STR[Pallet_2,Prdt_19KitKat,6].XPlace=P2_19KitKat_6_Place
;ENDFOLD
;FOLD OffsetPlace
Ponto_STR[Pallet_2,Prdt_19KitKat,6].OffsetPlace.X=0
Ponto_STR[Pallet_2,Prdt_19KitKat,6].OffsetPlace.Y=0
Ponto_STR[Pallet_2,Prdt_19KitKat,6].OffsetPlace.Z=0
Ponto_STR[Pallet_2,Prdt_19KitKat,6].OffsetPlace.A=0
Ponto_STR[Pallet_2,Prdt_19KitKat,6].OffsetPlace.B=0
Ponto_STR[Pallet_2,Prdt_19KitKat,6].OffsetPlace.C=0
;ENDFOLD
;ENDFOLD

;ENDFOLD
;FOLD LAYER 2: PLACE 7 ate 12
;FOLD PLACE 7
;FOLD PROPRIEDADES
Ponto_STR[Pallet_2,Prdt_19KitKat,7].NumCaixas = 1
Ponto_STR[Pallet_2,Prdt_19KitKat,7].PickOp = 1
Ponto_STR[Pallet_2,Prdt_19KitKat,7].ConfGarraOp = 0
Ponto_STR[Pallet_2,Prdt_19KitKat,7].FechaGarraOp = 0
Ponto_STR[Pallet_2,Prdt_19KitKat,7].AbreGarraOp = 0
Ponto_STR[Pallet_2,Prdt_19KitKat,7].SensoresCaixa = 1
Ponto_STR[Pallet_2,Prdt_19KitKat,7].TravaGarra = False
Ponto_STR[Pallet_2,Prdt_19KitKat,7].SkipGoHome = False
Ponto_STR[Pallet_2,Prdt_19KitKat,7].SkipSobeRelAtual = False
Ponto_STR[Pallet_2,Prdt_19KitKat,7].XApp1Place=P2_19KitKat_7_App1
Ponto_STR[Pallet_2,Prdt_19KitKat,7].XApp2Place=P2_19KitKat_7_App2
Ponto_STR[Pallet_2,Prdt_19KitKat,7].XPlace=P2_19KitKat_7_Place
;ENDFOLD
;FOLD OffsetPlace
Ponto_STR[Pallet_2,Prdt_19KitKat,7].OffsetPlace.X=0
Ponto_STR[Pallet_2,Prdt_19KitKat,7].OffsetPlace.Y=0
Ponto_STR[Pallet_2,Prdt_19KitKat,7].OffsetPlace.Z=0
Ponto_STR[Pallet_2,Prdt_19KitKat,7].OffsetPlace.A=0
Ponto_STR[Pallet_2,Prdt_19KitKat,7].OffsetPlace.B=0
Ponto_STR[Pallet_2,Prdt_19KitKat,7].OffsetPlace.C=0
;ENDFOLD
;ENDFOLD

;FOLD PLACE 8
;FOLD PROPRIEDADES
Ponto_STR[Pallet_2,Prdt_19KitKat,8].NumCaixas = 1
Ponto_STR[Pallet_2,Prdt_19KitKat,8].PickOp = 1
Ponto_STR[Pallet_2,Prdt_19KitKat,8].ConfGarraOp = 0
Ponto_STR[Pallet_2,Prdt_19KitKat,8].FechaGarraOp = 0
Ponto_STR[Pallet_2,Prdt_19KitKat,8].AbreGarraOp = 0
Ponto_STR[Pallet_2,Prdt_19KitKat,8].SensoresCaixa = 1
Ponto_STR[Pallet_2,Prdt_19KitKat,8].TravaGarra = False
Ponto_STR[Pallet_2,Prdt_19KitKat,8].SkipGoHome = False
Ponto_STR[Pallet_2,Prdt_19KitKat,8].SkipSobeRelAtual = False
Ponto_STR[Pallet_2,Prdt_19KitKat,8].XApp1Place=P2_19KitKat_8_App1
Ponto_STR[Pallet_2,Prdt_19KitKat,8].XApp2Place=P2_19KitKat_8_App2
Ponto_STR[Pallet_2,Prdt_19KitKat,8].XPlace=P2_19KitKat_8_Place
;ENDFOLD
;FOLD OffsetPlace
Ponto_STR[Pallet_2,Prdt_19KitKat,8].OffsetPlace.X=0
Ponto_STR[Pallet_2,Prdt_19KitKat,8].OffsetPlace.Y=0
Ponto_STR[Pallet_2,Prdt_19KitKat,8].OffsetPlace.Z=0
Ponto_STR[Pallet_2,Prdt_19KitKat,8].OffsetPlace.A=0
Ponto_STR[Pallet_2,Prdt_19KitKat,8].OffsetPlace.B=0
Ponto_STR[Pallet_2,Prdt_19KitKat,8].OffsetPlace.C=0
;ENDFOLD
;ENDFOLD

;FOLD PLACE 9
;FOLD PROPRIEDADES
Ponto_STR[Pallet_2,Prdt_19KitKat,9].NumCaixas = 1
Ponto_STR[Pallet_2,Prdt_19KitKat,9].PickOp = 1
Ponto_STR[Pallet_2,Prdt_19KitKat,9].ConfGarraOp = 0
Ponto_STR[Pallet_2,Prdt_19KitKat,9].FechaGarraOp = 0
Ponto_STR[Pallet_2,Prdt_19KitKat,9].AbreGarraOp = 0
Ponto_STR[Pallet_2,Prdt_19KitKat,9].SensoresCaixa = 1
Ponto_STR[Pallet_2,Prdt_19KitKat,9].TravaGarra = False
Ponto_STR[Pallet_2,Prdt_19KitKat,9].SkipGoHome = False
Ponto_STR[Pallet_2,Prdt_19KitKat,9].SkipSobeRelAtual = False
Ponto_STR[Pallet_2,Prdt_19KitKat,9].XApp1Place=P2_19KitKat_9_App1
Ponto_STR[Pallet_2,Prdt_19KitKat,9].XApp2Place=P2_19KitKat_9_App2
Ponto_STR[Pallet_2,Prdt_19KitKat,9].XPlace=P2_19KitKat_9_Place
;ENDFOLD
;FOLD OffsetPlace
Ponto_STR[Pallet_2,Prdt_19KitKat,9].OffsetPlace.X=0
Ponto_STR[Pallet_2,Prdt_19KitKat,9].OffsetPlace.Y=0
Ponto_STR[Pallet_2,Prdt_19KitKat,9].OffsetPlace.Z=0
Ponto_STR[Pallet_2,Prdt_19KitKat,9].OffsetPlace.A=0
Ponto_STR[Pallet_2,Prdt_19KitKat,9].OffsetPlace.B=0
Ponto_STR[Pallet_2,Prdt_19KitKat,9].OffsetPlace.C=0
;ENDFOLD
;ENDFOLD

;FOLD PLACE 10
;FOLD PROPRIEDADES
Ponto_STR[Pallet_2,Prdt_19KitKat,10].NumCaixas = 4
Ponto_STR[Pallet_2,Prdt_19KitKat,10].PickOp = 1
Ponto_STR[Pallet_2,Prdt_19KitKat,10].ConfGarraOp = 0
Ponto_STR[Pallet_2,Prdt_19KitKat,10].FechaGarraOp = 0
Ponto_STR[Pallet_2,Prdt_19KitKat,10].AbreGarraOp = 1
Ponto_STR[Pallet_2,Prdt_19KitKat,10].SensoresCaixa = 12345
Ponto_STR[Pallet_2,Prdt_19KitKat,10].TravaGarra = True
Ponto_STR[Pallet_2,Prdt_19KitKat,10].SkipGoHome = False
Ponto_STR[Pallet_2,Prdt_19KitKat,10].SkipSobeRelAtual = False
Ponto_STR[Pallet_2,Prdt_19KitKat,10].XApp1Place=P2_19KitKat_10_App1
Ponto_STR[Pallet_2,Prdt_19KitKat,10].XApp2Place=P2_19KitKat_10_App2
Ponto_STR[Pallet_2,Prdt_19KitKat,10].XPlace=P2_19KitKat_10_Place
;ENDFOLD
;FOLD OffsetPlace
Ponto_STR[Pallet_2,Prdt_19KitKat,10].OffsetPlace.X=0
Ponto_STR[Pallet_2,Prdt_19KitKat,10].OffsetPlace.Y=0
Ponto_STR[Pallet_2,Prdt_19KitKat,10].OffsetPlace.Z=0
Ponto_STR[Pallet_2,Prdt_19KitKat,10].OffsetPlace.A=0
Ponto_STR[Pallet_2,Prdt_19KitKat,10].OffsetPlace.B=0
Ponto_STR[Pallet_2,Prdt_19KitKat,10].OffsetPlace.C=0
;ENDFOLD
;ENDFOLD

;FOLD PLACE 11
;FOLD PROPRIEDADES
Ponto_STR[Pallet_2,Prdt_19KitKat,11].NumCaixas = 4
Ponto_STR[Pallet_2,Prdt_19KitKat,11].PickOp = 1
Ponto_STR[Pallet_2,Prdt_19KitKat,11].ConfGarraOp = 0
Ponto_STR[Pallet_2,Prdt_19KitKat,11].FechaGarraOp = 0
Ponto_STR[Pallet_2,Prdt_19KitKat,11].AbreGarraOp = 1
Ponto_STR[Pallet_2,Prdt_19KitKat,11].SensoresCaixa = 12345
Ponto_STR[Pallet_2,Prdt_19KitKat,11].TravaGarra = True
Ponto_STR[Pallet_2,Prdt_19KitKat,11].SkipGoHome = False
Ponto_STR[Pallet_2,Prdt_19KitKat,11].SkipSobeRelAtual = False
Ponto_STR[Pallet_2,Prdt_19KitKat,11].XApp1Place=P2_19KitKat_11_App1
Ponto_STR[Pallet_2,Prdt_19KitKat,11].XApp2Place=P2_19KitKat_11_App2
Ponto_STR[Pallet_2,Prdt_19KitKat,11].XPlace=P2_19KitKat_11_Place
;ENDFOLD
;FOLD OffsetPlace
Ponto_STR[Pallet_2,Prdt_19KitKat,11].OffsetPlace.X=0
Ponto_STR[Pallet_2,Prdt_19KitKat,11].OffsetPlace.Y=0
Ponto_STR[Pallet_2,Prdt_19KitKat,11].OffsetPlace.Z=0
Ponto_STR[Pallet_2,Prdt_19KitKat,11].OffsetPlace.A=0
Ponto_STR[Pallet_2,Prdt_19KitKat,11].OffsetPlace.B=0
Ponto_STR[Pallet_2,Prdt_19KitKat,11].OffsetPlace.C=0
;ENDFOLD
;ENDFOLD

;FOLD PLACE 12
;FOLD PROPRIEDADES
Ponto_STR[Pallet_2,Prdt_19KitKat,12].NumCaixas = 4
Ponto_STR[Pallet_2,Prdt_19KitKat,12].PickOp = 1
Ponto_STR[Pallet_2,Prdt_19KitKat,12].ConfGarraOp = 0
Ponto_STR[Pallet_2,Prdt_19KitKat,12].FechaGarraOp = 0
Ponto_STR[Pallet_2,Prdt_19KitKat,12].AbreGarraOp = 1
Ponto_STR[Pallet_2,Prdt_19KitKat,12].SensoresCaixa = 12345
Ponto_STR[Pallet_2,Prdt_19KitKat,12].TravaGarra = True
Ponto_STR[Pallet_2,Prdt_19KitKat,12].SkipGoHome = False
Ponto_STR[Pallet_2,Prdt_19KitKat,12].SkipSobeRelAtual = False
Ponto_STR[Pallet_2,Prdt_19KitKat,12].XApp1Place=P2_19KitKat_12_App1
Ponto_STR[Pallet_2,Prdt_19KitKat,12].XApp2Place=P2_19KitKat_12_App2
Ponto_STR[Pallet_2,Prdt_19KitKat,12].XPlace=P2_19KitKat_12_Place
;ENDFOLD
;FOLD OffsetPlace
Ponto_STR[Pallet_2,Prdt_19KitKat,12].OffsetPlace.X=0
Ponto_STR[Pallet_2,Prdt_19KitKat,12].OffsetPlace.Y=0
Ponto_STR[Pallet_2,Prdt_19KitKat,12].OffsetPlace.Z=0
Ponto_STR[Pallet_2,Prdt_19KitKat,12].OffsetPlace.A=0
Ponto_STR[Pallet_2,Prdt_19KitKat,12].OffsetPlace.B=0
Ponto_STR[Pallet_2,Prdt_19KitKat,12].OffsetPlace.C=0
;ENDFOLD
;ENDFOLD

;ENDFOLD
;ENDFOLD

;FOLD Pallet 2 - Produto 7Aero
;FOLD LAYER 1: PLACE 1 ate 8
;FOLD PLACE 1
;FOLD PROPRIEDADES
Ponto_STR[Pallet_2,Prdt_7Aero,1].NumCaixas = 3
Ponto_STR[Pallet_2,Prdt_7Aero,1].PickOp = 6
Ponto_STR[Pallet_2,Prdt_7Aero,1].ConfGarraOp = 0
Ponto_STR[Pallet_2,Prdt_7Aero,1].FechaGarraOp = 0
Ponto_STR[Pallet_2,Prdt_7Aero,1].AbreGarraOp = 0
Ponto_STR[Pallet_2,Prdt_7Aero,1].SensoresCaixa = 564
Ponto_STR[Pallet_2,Prdt_7Aero,1].TravaGarra = False
Ponto_STR[Pallet_2,Prdt_7Aero,1].SkipGoHome = False
Ponto_STR[Pallet_2,Prdt_7Aero,1].SkipSobeRelAtual = False
Ponto_STR[Pallet_2,Prdt_7Aero,1].XApp1Place=P2_7Aero_1_App1
Ponto_STR[Pallet_2,Prdt_7Aero,1].XApp2Place=P2_7Aero_1_App2
Ponto_STR[Pallet_2,Prdt_7Aero,1].XPlace=P2_7Aero_1_Place
;ENDFOLD
;FOLD OffsetPlace
Ponto_STR[Pallet_2,Prdt_7Aero,1].OffsetPlace.X=0
Ponto_STR[Pallet_2,Prdt_7Aero,1].OffsetPlace.Y=0
Ponto_STR[Pallet_2,Prdt_7Aero,1].OffsetPlace.Z=0
Ponto_STR[Pallet_2,Prdt_7Aero,1].OffsetPlace.A=0
Ponto_STR[Pallet_2,Prdt_7Aero,1].OffsetPlace.B=0
Ponto_STR[Pallet_2,Prdt_7Aero,1].OffsetPlace.C=0
;ENDFOLD
;ENDFOLD

;FOLD PLACE 2
;FOLD PROPRIEDADES
Ponto_STR[Pallet_2,Prdt_7Aero,2].NumCaixas = 3
Ponto_STR[Pallet_2,Prdt_7Aero,2].PickOp = 6
Ponto_STR[Pallet_2,Prdt_7Aero,2].ConfGarraOp = 0
Ponto_STR[Pallet_2,Prdt_7Aero,2].FechaGarraOp = 0
Ponto_STR[Pallet_2,Prdt_7Aero,2].AbreGarraOp = 0
Ponto_STR[Pallet_2,Prdt_7Aero,2].SensoresCaixa = 564
Ponto_STR[Pallet_2,Prdt_7Aero,2].TravaGarra = False
Ponto_STR[Pallet_2,Prdt_7Aero,2].SkipGoHome = False
Ponto_STR[Pallet_2,Prdt_7Aero,2].SkipSobeRelAtual = False
Ponto_STR[Pallet_2,Prdt_7Aero,2].XApp1Place=P2_7Aero_2_App1
Ponto_STR[Pallet_2,Prdt_7Aero,2].XApp2Place=P2_7Aero_2_App2
Ponto_STR[Pallet_2,Prdt_7Aero,2].XPlace=P2_7Aero_2_Place
;ENDFOLD
;FOLD OffsetPlace
Ponto_STR[Pallet_2,Prdt_7Aero,2].OffsetPlace.X=0
Ponto_STR[Pallet_2,Prdt_7Aero,2].OffsetPlace.Y=0
Ponto_STR[Pallet_2,Prdt_7Aero,2].OffsetPlace.Z=0
Ponto_STR[Pallet_2,Prdt_7Aero,2].OffsetPlace.A=0
Ponto_STR[Pallet_2,Prdt_7Aero,2].OffsetPlace.B=0
Ponto_STR[Pallet_2,Prdt_7Aero,2].OffsetPlace.C=0
;ENDFOLD
;ENDFOLD

;FOLD PLACE 3
;FOLD PROPRIEDADES
Ponto_STR[Pallet_2,Prdt_7Aero,3].NumCaixas = 2
Ponto_STR[Pallet_2,Prdt_7Aero,3].PickOp = 8
Ponto_STR[Pallet_2,Prdt_7Aero,3].ConfGarraOp = 5
Ponto_STR[Pallet_2,Prdt_7Aero,3].FechaGarraOp = 0
Ponto_STR[Pallet_2,Prdt_7Aero,3].AbreGarraOp = 0
Ponto_STR[Pallet_2,Prdt_7Aero,3].SensoresCaixa = 12
Ponto_STR[Pallet_2,Prdt_7Aero,3].TravaGarra = False
Ponto_STR[Pallet_2,Prdt_7Aero,3].SkipGoHome = False
Ponto_STR[Pallet_2,Prdt_7Aero,3].SkipSobeRelAtual = False
Ponto_STR[Pallet_2,Prdt_7Aero,3].XApp1Place=P2_7Aero_3_App1
Ponto_STR[Pallet_2,Prdt_7Aero,3].XApp2Place=P2_7Aero_3_App2
Ponto_STR[Pallet_2,Prdt_7Aero,3].XPlace=P2_7Aero_3_Place
;ENDFOLD
;FOLD OffsetPlace
Ponto_STR[Pallet_2,Prdt_7Aero,3].OffsetPlace.X=0
Ponto_STR[Pallet_2,Prdt_7Aero,3].OffsetPlace.Y=0
Ponto_STR[Pallet_2,Prdt_7Aero,3].OffsetPlace.Z=0
Ponto_STR[Pallet_2,Prdt_7Aero,3].OffsetPlace.A=0
Ponto_STR[Pallet_2,Prdt_7Aero,3].OffsetPlace.B=0
Ponto_STR[Pallet_2,Prdt_7Aero,3].OffsetPlace.C=0
;ENDFOLD
;ENDFOLD

;FOLD PLACE 4
;FOLD PROPRIEDADES
Ponto_STR[Pallet_2,Prdt_7Aero,4].NumCaixas = 2
Ponto_STR[Pallet_2,Prdt_7Aero,4].PickOp = 8
Ponto_STR[Pallet_2,Prdt_7Aero,4].ConfGarraOp = 5
Ponto_STR[Pallet_2,Prdt_7Aero,4].FechaGarraOp = 0
Ponto_STR[Pallet_2,Prdt_7Aero,4].AbreGarraOp = 0
Ponto_STR[Pallet_2,Prdt_7Aero,4].SensoresCaixa = 12
Ponto_STR[Pallet_2,Prdt_7Aero,4].TravaGarra = False
Ponto_STR[Pallet_2,Prdt_7Aero,4].SkipGoHome = False
Ponto_STR[Pallet_2,Prdt_7Aero,4].SkipSobeRelAtual = False
Ponto_STR[Pallet_2,Prdt_7Aero,4].XApp1Place=P2_7Aero_4_App1
Ponto_STR[Pallet_2,Prdt_7Aero,4].XApp2Place=P2_7Aero_4_App2
Ponto_STR[Pallet_2,Prdt_7Aero,4].XPlace=P2_7Aero_4_Place
;ENDFOLD
;FOLD OffsetPlace
Ponto_STR[Pallet_2,Prdt_7Aero,4].OffsetPlace.X=0
Ponto_STR[Pallet_2,Prdt_7Aero,4].OffsetPlace.Y=0
Ponto_STR[Pallet_2,Prdt_7Aero,4].OffsetPlace.Z=0
Ponto_STR[Pallet_2,Prdt_7Aero,4].OffsetPlace.A=0
Ponto_STR[Pallet_2,Prdt_7Aero,4].OffsetPlace.B=0
Ponto_STR[Pallet_2,Prdt_7Aero,4].OffsetPlace.C=0
;ENDFOLD
;ENDFOLD

;FOLD PLACE 5
;FOLD PROPRIEDADES
Ponto_STR[Pallet_2,Prdt_7Aero,5].NumCaixas = 3
Ponto_STR[Pallet_2,Prdt_7Aero,5].PickOp = 8
Ponto_STR[Pallet_2,Prdt_7Aero,5].ConfGarraOp = 5
Ponto_STR[Pallet_2,Prdt_7Aero,5].FechaGarraOp = 0
Ponto_STR[Pallet_2,Prdt_7Aero,5].AbreGarraOp = 1
Ponto_STR[Pallet_2,Prdt_7Aero,5].SensoresCaixa = 123
Ponto_STR[Pallet_2,Prdt_7Aero,5].TravaGarra = True
Ponto_STR[Pallet_2,Prdt_7Aero,5].SkipGoHome = False
Ponto_STR[Pallet_2,Prdt_7Aero,5].SkipSobeRelAtual = False
Ponto_STR[Pallet_2,Prdt_7Aero,5].XApp1Place=P2_7Aero_5_App1
Ponto_STR[Pallet_2,Prdt_7Aero,5].XApp2Place=P2_7Aero_5_App2
Ponto_STR[Pallet_2,Prdt_7Aero,5].XPlace=P2_7Aero_5_Place
;ENDFOLD
;FOLD OffsetPlace
Ponto_STR[Pallet_2,Prdt_7Aero,5].OffsetPlace.X=0
Ponto_STR[Pallet_2,Prdt_7Aero,5].OffsetPlace.Y=0
Ponto_STR[Pallet_2,Prdt_7Aero,5].OffsetPlace.Z=0
Ponto_STR[Pallet_2,Prdt_7Aero,5].OffsetPlace.A=0
Ponto_STR[Pallet_2,Prdt_7Aero,5].OffsetPlace.B=0
Ponto_STR[Pallet_2,Prdt_7Aero,5].OffsetPlace.C=0
;ENDFOLD
;ENDFOLD

;FOLD PLACE 6
;FOLD PROPRIEDADES
Ponto_STR[Pallet_2,Prdt_7Aero,6].NumCaixas = 3
Ponto_STR[Pallet_2,Prdt_7Aero,6].PickOp = 8
Ponto_STR[Pallet_2,Prdt_7Aero,6].ConfGarraOp = 5
Ponto_STR[Pallet_2,Prdt_7Aero,6].FechaGarraOp = 0
Ponto_STR[Pallet_2,Prdt_7Aero,6].AbreGarraOp = 1
Ponto_STR[Pallet_2,Prdt_7Aero,6].SensoresCaixa = 123
Ponto_STR[Pallet_2,Prdt_7Aero,6].TravaGarra = True
Ponto_STR[Pallet_2,Prdt_7Aero,6].SkipGoHome = False
Ponto_STR[Pallet_2,Prdt_7Aero,6].SkipSobeRelAtual = False
Ponto_STR[Pallet_2,Prdt_7Aero,6].XApp1Place=P2_7Aero_6_App1
Ponto_STR[Pallet_2,Prdt_7Aero,6].XApp2Place=P2_7Aero_6_App2
Ponto_STR[Pallet_2,Prdt_7Aero,6].XPlace=P2_7Aero_6_Place
;ENDFOLD
;FOLD OffsetPlace
Ponto_STR[Pallet_2,Prdt_7Aero,6].OffsetPlace.X=0
Ponto_STR[Pallet_2,Prdt_7Aero,6].OffsetPlace.Y=0
Ponto_STR[Pallet_2,Prdt_7Aero,6].OffsetPlace.Z=0
Ponto_STR[Pallet_2,Prdt_7Aero,6].OffsetPlace.A=0
Ponto_STR[Pallet_2,Prdt_7Aero,6].OffsetPlace.B=0
Ponto_STR[Pallet_2,Prdt_7Aero,6].OffsetPlace.C=0
;ENDFOLD
;ENDFOLD

;FOLD PLACE 7
;FOLD PROPRIEDADES
Ponto_STR[Pallet_2,Prdt_7Aero,7].NumCaixas = 2
Ponto_STR[Pallet_2,Prdt_7Aero,7].PickOp = 8
Ponto_STR[Pallet_2,Prdt_7Aero,7].ConfGarraOp = 5
Ponto_STR[Pallet_2,Prdt_7Aero,7].FechaGarraOp = 0
Ponto_STR[Pallet_2,Prdt_7Aero,7].AbreGarraOp = 1
Ponto_STR[Pallet_2,Prdt_7Aero,7].SensoresCaixa = 12
Ponto_STR[Pallet_2,Prdt_7Aero,7].TravaGarra = True
Ponto_STR[Pallet_2,Prdt_7Aero,7].SkipGoHome = False
Ponto_STR[Pallet_2,Prdt_7Aero,7].SkipSobeRelAtual = False
Ponto_STR[Pallet_2,Prdt_7Aero,7].XApp1Place=P2_7Aero_7_App1
Ponto_STR[Pallet_2,Prdt_7Aero,7].XApp2Place=P2_7Aero_7_App2
Ponto_STR[Pallet_2,Prdt_7Aero,7].XPlace=P2_7Aero_7_Place
;ENDFOLD
;FOLD OffsetPlace
Ponto_STR[Pallet_2,Prdt_7Aero,7].OffsetPlace.X=0
Ponto_STR[Pallet_2,Prdt_7Aero,7].OffsetPlace.Y=0
Ponto_STR[Pallet_2,Prdt_7Aero,7].OffsetPlace.Z=0
Ponto_STR[Pallet_2,Prdt_7Aero,7].OffsetPlace.A=0
Ponto_STR[Pallet_2,Prdt_7Aero,7].OffsetPlace.B=0
Ponto_STR[Pallet_2,Prdt_7Aero,7].OffsetPlace.C=0
;ENDFOLD
;ENDFOLD

;FOLD PLACE 8
;FOLD PROPRIEDADES
Ponto_STR[Pallet_2,Prdt_7Aero,8].NumCaixas = 2
Ponto_STR[Pallet_2,Prdt_7Aero,8].PickOp = 8
Ponto_STR[Pallet_2,Prdt_7Aero,8].ConfGarraOp = 5
Ponto_STR[Pallet_2,Prdt_7Aero,8].FechaGarraOp = 0
Ponto_STR[Pallet_2,Prdt_7Aero,8].AbreGarraOp = 1
Ponto_STR[Pallet_2,Prdt_7Aero,8].SensoresCaixa = 12
Ponto_STR[Pallet_2,Prdt_7Aero,8].TravaGarra = True
Ponto_STR[Pallet_2,Prdt_7Aero,8].SkipGoHome = False
Ponto_STR[Pallet_2,Prdt_7Aero,8].SkipSobeRelAtual = False
Ponto_STR[Pallet_2,Prdt_7Aero,8].XApp1Place=P2_7Aero_8_App1
Ponto_STR[Pallet_2,Prdt_7Aero,8].XApp2Place=P2_7Aero_8_App2
Ponto_STR[Pallet_2,Prdt_7Aero,8].XPlace=P2_7Aero_8_Place
;ENDFOLD
;FOLD OffsetPlace
Ponto_STR[Pallet_2,Prdt_7Aero,8].OffsetPlace.X=0
Ponto_STR[Pallet_2,Prdt_7Aero,8].OffsetPlace.Y=0
Ponto_STR[Pallet_2,Prdt_7Aero,8].OffsetPlace.Z=0
Ponto_STR[Pallet_2,Prdt_7Aero,8].OffsetPlace.A=0
Ponto_STR[Pallet_2,Prdt_7Aero,8].OffsetPlace.B=0
Ponto_STR[Pallet_2,Prdt_7Aero,8].OffsetPlace.C=0
;ENDFOLD
;ENDFOLD

;ENDFOLD
;FOLD LAYER 2: PLACE 9 ate 16
;FOLD PLACE 9
;FOLD PROPRIEDADES
Ponto_STR[Pallet_2,Prdt_7Aero,9].NumCaixas = 2
Ponto_STR[Pallet_2,Prdt_7Aero,9].PickOp = 8
Ponto_STR[Pallet_2,Prdt_7Aero,9].ConfGarraOp = 5
Ponto_STR[Pallet_2,Prdt_7Aero,9].FechaGarraOp = 0
Ponto_STR[Pallet_2,Prdt_7Aero,9].AbreGarraOp = 1
Ponto_STR[Pallet_2,Prdt_7Aero,9].SensoresCaixa = 12
Ponto_STR[Pallet_2,Prdt_7Aero,9].TravaGarra = True
Ponto_STR[Pallet_2,Prdt_7Aero,9].SkipGoHome = False
Ponto_STR[Pallet_2,Prdt_7Aero,9].SkipSobeRelAtual = False
Ponto_STR[Pallet_2,Prdt_7Aero,9].XApp1Place=P2_7Aero_9_App1
Ponto_STR[Pallet_2,Prdt_7Aero,9].XApp2Place=P2_7Aero_9_App2
Ponto_STR[Pallet_2,Prdt_7Aero,9].XPlace=P2_7Aero_9_Place
;ENDFOLD
;FOLD OffsetPlace
Ponto_STR[Pallet_2,Prdt_7Aero,9].OffsetPlace.X=0
Ponto_STR[Pallet_2,Prdt_7Aero,9].OffsetPlace.Y=0
Ponto_STR[Pallet_2,Prdt_7Aero,9].OffsetPlace.Z=0
Ponto_STR[Pallet_2,Prdt_7Aero,9].OffsetPlace.A=0
Ponto_STR[Pallet_2,Prdt_7Aero,9].OffsetPlace.B=0
Ponto_STR[Pallet_2,Prdt_7Aero,9].OffsetPlace.C=0
;ENDFOLD
;ENDFOLD

;FOLD PLACE 10
;FOLD PROPRIEDADES
Ponto_STR[Pallet_2,Prdt_7Aero,10].NumCaixas = 2
Ponto_STR[Pallet_2,Prdt_7Aero,10].PickOp = 8
Ponto_STR[Pallet_2,Prdt_7Aero,10].ConfGarraOp = 5
Ponto_STR[Pallet_2,Prdt_7Aero,10].FechaGarraOp = 0
Ponto_STR[Pallet_2,Prdt_7Aero,10].AbreGarraOp = 1
Ponto_STR[Pallet_2,Prdt_7Aero,10].SensoresCaixa = 12
Ponto_STR[Pallet_2,Prdt_7Aero,10].TravaGarra = True
Ponto_STR[Pallet_2,Prdt_7Aero,10].SkipGoHome = False
Ponto_STR[Pallet_2,Prdt_7Aero,10].SkipSobeRelAtual = False
Ponto_STR[Pallet_2,Prdt_7Aero,10].XApp1Place=P2_7Aero_10_App1
Ponto_STR[Pallet_2,Prdt_7Aero,10].XApp2Place=P2_7Aero_10_App2
Ponto_STR[Pallet_2,Prdt_7Aero,10].XPlace=P2_7Aero_10_Place
;ENDFOLD
;FOLD OffsetPlace
Ponto_STR[Pallet_2,Prdt_7Aero,10].OffsetPlace.X=0
Ponto_STR[Pallet_2,Prdt_7Aero,10].OffsetPlace.Y=0
Ponto_STR[Pallet_2,Prdt_7Aero,10].OffsetPlace.Z=0
Ponto_STR[Pallet_2,Prdt_7Aero,10].OffsetPlace.A=0
Ponto_STR[Pallet_2,Prdt_7Aero,10].OffsetPlace.B=0
Ponto_STR[Pallet_2,Prdt_7Aero,10].OffsetPlace.C=0
;ENDFOLD
;ENDFOLD

;FOLD PLACE 11
;FOLD PROPRIEDADES
Ponto_STR[Pallet_2,Prdt_7Aero,11].NumCaixas = 3
Ponto_STR[Pallet_2,Prdt_7Aero,11].PickOp = 8
Ponto_STR[Pallet_2,Prdt_7Aero,11].ConfGarraOp = 5
Ponto_STR[Pallet_2,Prdt_7Aero,11].FechaGarraOp = 0
Ponto_STR[Pallet_2,Prdt_7Aero,11].AbreGarraOp = 0
Ponto_STR[Pallet_2,Prdt_7Aero,11].SensoresCaixa = 123
Ponto_STR[Pallet_2,Prdt_7Aero,11].TravaGarra = False
Ponto_STR[Pallet_2,Prdt_7Aero,11].SkipGoHome = False
Ponto_STR[Pallet_2,Prdt_7Aero,11].SkipSobeRelAtual = False
Ponto_STR[Pallet_2,Prdt_7Aero,11].XApp1Place=P2_7Aero_11_App1
Ponto_STR[Pallet_2,Prdt_7Aero,11].XApp2Place=P2_7Aero_11_App2
Ponto_STR[Pallet_2,Prdt_7Aero,11].XPlace=P2_7Aero_11_Place
;ENDFOLD
;FOLD OffsetPlace
Ponto_STR[Pallet_2,Prdt_7Aero,11].OffsetPlace.X=0
Ponto_STR[Pallet_2,Prdt_7Aero,11].OffsetPlace.Y=0
Ponto_STR[Pallet_2,Prdt_7Aero,11].OffsetPlace.Z=0
Ponto_STR[Pallet_2,Prdt_7Aero,11].OffsetPlace.A=0
Ponto_STR[Pallet_2,Prdt_7Aero,11].OffsetPlace.B=0
Ponto_STR[Pallet_2,Prdt_7Aero,11].OffsetPlace.C=0
;ENDFOLD
;ENDFOLD

;FOLD PLACE 12
;FOLD PROPRIEDADES
Ponto_STR[Pallet_2,Prdt_7Aero,12].NumCaixas = 3
Ponto_STR[Pallet_2,Prdt_7Aero,12].PickOp = 8
Ponto_STR[Pallet_2,Prdt_7Aero,12].ConfGarraOp = 5
Ponto_STR[Pallet_2,Prdt_7Aero,12].FechaGarraOp = 0
Ponto_STR[Pallet_2,Prdt_7Aero,12].AbreGarraOp = 0
Ponto_STR[Pallet_2,Prdt_7Aero,12].SensoresCaixa = 123
Ponto_STR[Pallet_2,Prdt_7Aero,12].TravaGarra = False
Ponto_STR[Pallet_2,Prdt_7Aero,12].SkipGoHome = False
Ponto_STR[Pallet_2,Prdt_7Aero,12].SkipSobeRelAtual = False
Ponto_STR[Pallet_2,Prdt_7Aero,12].XApp1Place=P2_7Aero_12_App1
Ponto_STR[Pallet_2,Prdt_7Aero,12].XApp2Place=P2_7Aero_12_App2
Ponto_STR[Pallet_2,Prdt_7Aero,12].XPlace=P2_7Aero_12_Place
;ENDFOLD
;FOLD OffsetPlace
Ponto_STR[Pallet_2,Prdt_7Aero,12].OffsetPlace.X=0
Ponto_STR[Pallet_2,Prdt_7Aero,12].OffsetPlace.Y=0
Ponto_STR[Pallet_2,Prdt_7Aero,12].OffsetPlace.Z=0
Ponto_STR[Pallet_2,Prdt_7Aero,12].OffsetPlace.A=0
Ponto_STR[Pallet_2,Prdt_7Aero,12].OffsetPlace.B=0
Ponto_STR[Pallet_2,Prdt_7Aero,12].OffsetPlace.C=0
;ENDFOLD
;ENDFOLD

;FOLD PLACE 13
;FOLD PROPRIEDADES
Ponto_STR[Pallet_2,Prdt_7Aero,13].NumCaixas = 3
Ponto_STR[Pallet_2,Prdt_7Aero,13].PickOp = 8
Ponto_STR[Pallet_2,Prdt_7Aero,13].ConfGarraOp = 5
Ponto_STR[Pallet_2,Prdt_7Aero,13].FechaGarraOp = 0
Ponto_STR[Pallet_2,Prdt_7Aero,13].AbreGarraOp = 0
Ponto_STR[Pallet_2,Prdt_7Aero,13].SensoresCaixa = 123
Ponto_STR[Pallet_2,Prdt_7Aero,13].TravaGarra = False
Ponto_STR[Pallet_2,Prdt_7Aero,13].SkipGoHome = False
Ponto_STR[Pallet_2,Prdt_7Aero,13].SkipSobeRelAtual = False
Ponto_STR[Pallet_2,Prdt_7Aero,13].XApp1Place=P2_7Aero_13_App1
Ponto_STR[Pallet_2,Prdt_7Aero,13].XApp2Place=P2_7Aero_13_App2
Ponto_STR[Pallet_2,Prdt_7Aero,13].XPlace=P2_7Aero_13_Place
;ENDFOLD
;FOLD OffsetPlace
Ponto_STR[Pallet_2,Prdt_7Aero,13].OffsetPlace.X=0
Ponto_STR[Pallet_2,Prdt_7Aero,13].OffsetPlace.Y=0
Ponto_STR[Pallet_2,Prdt_7Aero,13].OffsetPlace.Z=0
Ponto_STR[Pallet_2,Prdt_7Aero,13].OffsetPlace.A=0
Ponto_STR[Pallet_2,Prdt_7Aero,13].OffsetPlace.B=0
Ponto_STR[Pallet_2,Prdt_7Aero,13].OffsetPlace.C=0
;ENDFOLD
;ENDFOLD

;FOLD PLACE 14
;FOLD PROPRIEDADES
Ponto_STR[Pallet_2,Prdt_7Aero,14].NumCaixas = 3
Ponto_STR[Pallet_2,Prdt_7Aero,14].PickOp = 8
Ponto_STR[Pallet_2,Prdt_7Aero,14].ConfGarraOp = 5
Ponto_STR[Pallet_2,Prdt_7Aero,14].FechaGarraOp = 0
Ponto_STR[Pallet_2,Prdt_7Aero,14].AbreGarraOp = 0
Ponto_STR[Pallet_2,Prdt_7Aero,14].SensoresCaixa = 123
Ponto_STR[Pallet_2,Prdt_7Aero,14].TravaGarra = False
Ponto_STR[Pallet_2,Prdt_7Aero,14].SkipGoHome = False
Ponto_STR[Pallet_2,Prdt_7Aero,14].SkipSobeRelAtual = False
Ponto_STR[Pallet_2,Prdt_7Aero,14].XApp1Place=P2_7Aero_14_App1
Ponto_STR[Pallet_2,Prdt_7Aero,14].XApp2Place=P2_7Aero_14_App2
Ponto_STR[Pallet_2,Prdt_7Aero,14].XPlace=P2_7Aero_14_Place
;ENDFOLD
;FOLD OffsetPlace
Ponto_STR[Pallet_2,Prdt_7Aero,14].OffsetPlace.X=0
Ponto_STR[Pallet_2,Prdt_7Aero,14].OffsetPlace.Y=0
Ponto_STR[Pallet_2,Prdt_7Aero,14].OffsetPlace.Z=0
Ponto_STR[Pallet_2,Prdt_7Aero,14].OffsetPlace.A=0
Ponto_STR[Pallet_2,Prdt_7Aero,14].OffsetPlace.B=0
Ponto_STR[Pallet_2,Prdt_7Aero,14].OffsetPlace.C=0
;ENDFOLD
;ENDFOLD

;FOLD PLACE 15
;FOLD PROPRIEDADES
Ponto_STR[Pallet_2,Prdt_7Aero,15].NumCaixas = 2
Ponto_STR[Pallet_2,Prdt_7Aero,15].PickOp = 8
Ponto_STR[Pallet_2,Prdt_7Aero,15].ConfGarraOp = 5
Ponto_STR[Pallet_2,Prdt_7Aero,15].FechaGarraOp = 0
Ponto_STR[Pallet_2,Prdt_7Aero,15].AbreGarraOp = 1
Ponto_STR[Pallet_2,Prdt_7Aero,15].SensoresCaixa = 12
Ponto_STR[Pallet_2,Prdt_7Aero,15].TravaGarra = True
Ponto_STR[Pallet_2,Prdt_7Aero,15].SkipGoHome = False
Ponto_STR[Pallet_2,Prdt_7Aero,15].SkipSobeRelAtual = False
Ponto_STR[Pallet_2,Prdt_7Aero,15].XApp1Place=P2_7Aero_15_App1
Ponto_STR[Pallet_2,Prdt_7Aero,15].XApp2Place=P2_7Aero_15_App2
Ponto_STR[Pallet_2,Prdt_7Aero,15].XPlace=P2_7Aero_15_Place
;ENDFOLD
;FOLD OffsetPlace
Ponto_STR[Pallet_2,Prdt_7Aero,15].OffsetPlace.X=0
Ponto_STR[Pallet_2,Prdt_7Aero,15].OffsetPlace.Y=0
Ponto_STR[Pallet_2,Prdt_7Aero,15].OffsetPlace.Z=0
Ponto_STR[Pallet_2,Prdt_7Aero,15].OffsetPlace.A=0
Ponto_STR[Pallet_2,Prdt_7Aero,15].OffsetPlace.B=0
Ponto_STR[Pallet_2,Prdt_7Aero,15].OffsetPlace.C=0
;ENDFOLD
;ENDFOLD

;FOLD PLACE 16
;FOLD PROPRIEDADES
Ponto_STR[Pallet_2,Prdt_7Aero,16].NumCaixas = 2
Ponto_STR[Pallet_2,Prdt_7Aero,16].PickOp = 8
Ponto_STR[Pallet_2,Prdt_7Aero,16].ConfGarraOp = 5
Ponto_STR[Pallet_2,Prdt_7Aero,16].FechaGarraOp = 0
Ponto_STR[Pallet_2,Prdt_7Aero,16].AbreGarraOp = 1
Ponto_STR[Pallet_2,Prdt_7Aero,16].SensoresCaixa = 12
Ponto_STR[Pallet_2,Prdt_7Aero,16].TravaGarra = True
Ponto_STR[Pallet_2,Prdt_7Aero,16].SkipGoHome = False
Ponto_STR[Pallet_2,Prdt_7Aero,16].SkipSobeRelAtual = False
Ponto_STR[Pallet_2,Prdt_7Aero,16].XApp1Place=P2_7Aero_16_App1
Ponto_STR[Pallet_2,Prdt_7Aero,16].XApp2Place=P2_7Aero_16_App2
Ponto_STR[Pallet_2,Prdt_7Aero,16].XPlace=P2_7Aero_16_Place
;ENDFOLD
;FOLD OffsetPlace
Ponto_STR[Pallet_2,Prdt_7Aero,16].OffsetPlace.X=0
Ponto_STR[Pallet_2,Prdt_7Aero,16].OffsetPlace.Y=0
Ponto_STR[Pallet_2,Prdt_7Aero,16].OffsetPlace.Z=0
Ponto_STR[Pallet_2,Prdt_7Aero,16].OffsetPlace.A=0
Ponto_STR[Pallet_2,Prdt_7Aero,16].OffsetPlace.B=0
Ponto_STR[Pallet_2,Prdt_7Aero,16].OffsetPlace.C=0
;ENDFOLD
;ENDFOLD

;ENDFOLD
;ENDFOLD

;FOLD Pallet 2 - Produto 15CoffeCrisp
;FOLD LAYER 1: PLACE 1 ate 7
;FOLD PLACE 1
;FOLD PROPRIEDADES
Ponto_STR[Pallet_2,Prdt_15CoffeCrisp,1].NumCaixas = 1
Ponto_STR[Pallet_2,Prdt_15CoffeCrisp,1].PickOp = 8
Ponto_STR[Pallet_2,Prdt_15CoffeCrisp,1].ConfGarraOp = 5
Ponto_STR[Pallet_2,Prdt_15CoffeCrisp,1].FechaGarraOp = 0
Ponto_STR[Pallet_2,Prdt_15CoffeCrisp,1].AbreGarraOp = 0
Ponto_STR[Pallet_2,Prdt_15CoffeCrisp,1].SensoresCaixa = 1
Ponto_STR[Pallet_2,Prdt_15CoffeCrisp,1].TravaGarra = False
Ponto_STR[Pallet_2,Prdt_15CoffeCrisp,1].SkipGoHome = False
Ponto_STR[Pallet_2,Prdt_15CoffeCrisp,1].SkipSobeRelAtual = False
Ponto_STR[Pallet_2,Prdt_15CoffeCrisp,1].XApp1Place=P2_15CoffeCrisp_1_App1
Ponto_STR[Pallet_2,Prdt_15CoffeCrisp,1].XApp2Place=P2_15CoffeCrisp_1_App2
Ponto_STR[Pallet_2,Prdt_15CoffeCrisp,1].XPlace=P2_15CoffeCrisp_1_Place
;ENDFOLD
;FOLD OffsetPlace
Ponto_STR[Pallet_2,Prdt_15CoffeCrisp,1].OffsetPlace.X=0
Ponto_STR[Pallet_2,Prdt_15CoffeCrisp,1].OffsetPlace.Y=0
Ponto_STR[Pallet_2,Prdt_15CoffeCrisp,1].OffsetPlace.Z=0
Ponto_STR[Pallet_2,Prdt_15CoffeCrisp,1].OffsetPlace.A=0
Ponto_STR[Pallet_2,Prdt_15CoffeCrisp,1].OffsetPlace.B=0
Ponto_STR[Pallet_2,Prdt_15CoffeCrisp,1].OffsetPlace.C=0
;ENDFOLD
;ENDFOLD

;FOLD PLACE 2
;FOLD PROPRIEDADES
Ponto_STR[Pallet_2,Prdt_15CoffeCrisp,2].NumCaixas = 1
Ponto_STR[Pallet_2,Prdt_15CoffeCrisp,2].PickOp = 8
Ponto_STR[Pallet_2,Prdt_15CoffeCrisp,2].ConfGarraOp = 5
Ponto_STR[Pallet_2,Prdt_15CoffeCrisp,2].FechaGarraOp = 0
Ponto_STR[Pallet_2,Prdt_15CoffeCrisp,2].AbreGarraOp = 0
Ponto_STR[Pallet_2,Prdt_15CoffeCrisp,2].SensoresCaixa = 1
Ponto_STR[Pallet_2,Prdt_15CoffeCrisp,2].TravaGarra = False
Ponto_STR[Pallet_2,Prdt_15CoffeCrisp,2].SkipGoHome = False
Ponto_STR[Pallet_2,Prdt_15CoffeCrisp,2].SkipSobeRelAtual = False
Ponto_STR[Pallet_2,Prdt_15CoffeCrisp,2].XApp1Place=P2_15CoffeCrisp_2_App1
Ponto_STR[Pallet_2,Prdt_15CoffeCrisp,2].XApp2Place=P2_15CoffeCrisp_2_App2
Ponto_STR[Pallet_2,Prdt_15CoffeCrisp,2].XPlace=P2_15CoffeCrisp_2_Place
;ENDFOLD
;FOLD OffsetPlace
Ponto_STR[Pallet_2,Prdt_15CoffeCrisp,2].OffsetPlace.X=0
Ponto_STR[Pallet_2,Prdt_15CoffeCrisp,2].OffsetPlace.Y=0
Ponto_STR[Pallet_2,Prdt_15CoffeCrisp,2].OffsetPlace.Z=0
Ponto_STR[Pallet_2,Prdt_15CoffeCrisp,2].OffsetPlace.A=0
Ponto_STR[Pallet_2,Prdt_15CoffeCrisp,2].OffsetPlace.B=0
Ponto_STR[Pallet_2,Prdt_15CoffeCrisp,2].OffsetPlace.C=0
;ENDFOLD
;ENDFOLD

;FOLD PLACE 3
;FOLD PROPRIEDADES
Ponto_STR[Pallet_2,Prdt_15CoffeCrisp,3].NumCaixas = 1
Ponto_STR[Pallet_2,Prdt_15CoffeCrisp,3].PickOp = 8
Ponto_STR[Pallet_2,Prdt_15CoffeCrisp,3].ConfGarraOp = 5
Ponto_STR[Pallet_2,Prdt_15CoffeCrisp,3].FechaGarraOp = 0
Ponto_STR[Pallet_2,Prdt_15CoffeCrisp,3].AbreGarraOp = 0
Ponto_STR[Pallet_2,Prdt_15CoffeCrisp,3].SensoresCaixa = 1
Ponto_STR[Pallet_2,Prdt_15CoffeCrisp,3].TravaGarra = False
Ponto_STR[Pallet_2,Prdt_15CoffeCrisp,3].SkipGoHome = False
Ponto_STR[Pallet_2,Prdt_15CoffeCrisp,3].SkipSobeRelAtual = False
Ponto_STR[Pallet_2,Prdt_15CoffeCrisp,3].XApp1Place=P2_15CoffeCrisp_3_App1
Ponto_STR[Pallet_2,Prdt_15CoffeCrisp,3].XApp2Place=P2_15CoffeCrisp_3_App2
Ponto_STR[Pallet_2,Prdt_15CoffeCrisp,3].XPlace=P2_15CoffeCrisp_3_Place
;ENDFOLD
;FOLD OffsetPlace
Ponto_STR[Pallet_2,Prdt_15CoffeCrisp,3].OffsetPlace.X=0
Ponto_STR[Pallet_2,Prdt_15CoffeCrisp,3].OffsetPlace.Y=0
Ponto_STR[Pallet_2,Prdt_15CoffeCrisp,3].OffsetPlace.Z=0
Ponto_STR[Pallet_2,Prdt_15CoffeCrisp,3].OffsetPlace.A=0
Ponto_STR[Pallet_2,Prdt_15CoffeCrisp,3].OffsetPlace.B=0
Ponto_STR[Pallet_2,Prdt_15CoffeCrisp,3].OffsetPlace.C=0
;ENDFOLD
;ENDFOLD

;FOLD PLACE 4
;FOLD PROPRIEDADES
Ponto_STR[Pallet_2,Prdt_15CoffeCrisp,4].NumCaixas = 2
Ponto_STR[Pallet_2,Prdt_15CoffeCrisp,4].PickOp = 8
Ponto_STR[Pallet_2,Prdt_15CoffeCrisp,4].ConfGarraOp = 5
Ponto_STR[Pallet_2,Prdt_15CoffeCrisp,4].FechaGarraOp = 0
Ponto_STR[Pallet_2,Prdt_15CoffeCrisp,4].AbreGarraOp = 1
Ponto_STR[Pallet_2,Prdt_15CoffeCrisp,4].SensoresCaixa = 123
Ponto_STR[Pallet_2,Prdt_15CoffeCrisp,4].TravaGarra = True
Ponto_STR[Pallet_2,Prdt_15CoffeCrisp,4].SkipGoHome = False
Ponto_STR[Pallet_2,Prdt_15CoffeCrisp,4].SkipSobeRelAtual = False
Ponto_STR[Pallet_2,Prdt_15CoffeCrisp,4].XApp1Place=P2_15CoffeCrisp_4_App1
Ponto_STR[Pallet_2,Prdt_15CoffeCrisp,4].XApp2Place=P2_15CoffeCrisp_4_App2
Ponto_STR[Pallet_2,Prdt_15CoffeCrisp,4].XPlace=P2_15CoffeCrisp_4_Place
;ENDFOLD
;FOLD OffsetPlace
Ponto_STR[Pallet_2,Prdt_15CoffeCrisp,4].OffsetPlace.X=0
Ponto_STR[Pallet_2,Prdt_15CoffeCrisp,4].OffsetPlace.Y=0
Ponto_STR[Pallet_2,Prdt_15CoffeCrisp,4].OffsetPlace.Z=0
Ponto_STR[Pallet_2,Prdt_15CoffeCrisp,4].OffsetPlace.A=0
Ponto_STR[Pallet_2,Prdt_15CoffeCrisp,4].OffsetPlace.B=0
Ponto_STR[Pallet_2,Prdt_15CoffeCrisp,4].OffsetPlace.C=0
;ENDFOLD
;ENDFOLD

;FOLD PLACE 5
;FOLD PROPRIEDADES
Ponto_STR[Pallet_2,Prdt_15CoffeCrisp,5].NumCaixas = 2
Ponto_STR[Pallet_2,Prdt_15CoffeCrisp,5].PickOp = 8
Ponto_STR[Pallet_2,Prdt_15CoffeCrisp,5].ConfGarraOp = 5
Ponto_STR[Pallet_2,Prdt_15CoffeCrisp,5].FechaGarraOp = 0
Ponto_STR[Pallet_2,Prdt_15CoffeCrisp,5].AbreGarraOp = 1
Ponto_STR[Pallet_2,Prdt_15CoffeCrisp,5].SensoresCaixa = 123
Ponto_STR[Pallet_2,Prdt_15CoffeCrisp,5].TravaGarra = True
Ponto_STR[Pallet_2,Prdt_15CoffeCrisp,5].SkipGoHome = False
Ponto_STR[Pallet_2,Prdt_15CoffeCrisp,5].SkipSobeRelAtual = False
Ponto_STR[Pallet_2,Prdt_15CoffeCrisp,5].XApp1Place=P2_15CoffeCrisp_5_App1
Ponto_STR[Pallet_2,Prdt_15CoffeCrisp,5].XApp2Place=P2_15CoffeCrisp_5_App2
Ponto_STR[Pallet_2,Prdt_15CoffeCrisp,5].XPlace=P2_15CoffeCrisp_5_Place
;ENDFOLD
;FOLD OffsetPlace
Ponto_STR[Pallet_2,Prdt_15CoffeCrisp,5].OffsetPlace.X=0
Ponto_STR[Pallet_2,Prdt_15CoffeCrisp,5].OffsetPlace.Y=0
Ponto_STR[Pallet_2,Prdt_15CoffeCrisp,5].OffsetPlace.Z=0
Ponto_STR[Pallet_2,Prdt_15CoffeCrisp,5].OffsetPlace.A=0
Ponto_STR[Pallet_2,Prdt_15CoffeCrisp,5].OffsetPlace.B=0
Ponto_STR[Pallet_2,Prdt_15CoffeCrisp,5].OffsetPlace.C=0
;ENDFOLD
;ENDFOLD

;FOLD PLACE 6
;FOLD PROPRIEDADES
Ponto_STR[Pallet_2,Prdt_15CoffeCrisp,6].NumCaixas = 3
Ponto_STR[Pallet_2,Prdt_15CoffeCrisp,6].PickOp = 8
Ponto_STR[Pallet_2,Prdt_15CoffeCrisp,6].ConfGarraOp = 5
Ponto_STR[Pallet_2,Prdt_15CoffeCrisp,6].FechaGarraOp = 0
Ponto_STR[Pallet_2,Prdt_15CoffeCrisp,6].AbreGarraOp = 0
Ponto_STR[Pallet_2,Prdt_15CoffeCrisp,6].SensoresCaixa = 1234
Ponto_STR[Pallet_2,Prdt_15CoffeCrisp,6].TravaGarra = False
Ponto_STR[Pallet_2,Prdt_15CoffeCrisp,6].SkipGoHome = False
Ponto_STR[Pallet_2,Prdt_15CoffeCrisp,6].SkipSobeRelAtual = False
Ponto_STR[Pallet_2,Prdt_15CoffeCrisp,6].XApp1Place=P2_15CoffeCrisp_6_App1
Ponto_STR[Pallet_2,Prdt_15CoffeCrisp,6].XApp2Place=P2_15CoffeCrisp_6_App2
Ponto_STR[Pallet_2,Prdt_15CoffeCrisp,6].XPlace=P2_15CoffeCrisp_6_Place
;ENDFOLD
;FOLD OffsetPlace
Ponto_STR[Pallet_2,Prdt_15CoffeCrisp,6].OffsetPlace.X=0
Ponto_STR[Pallet_2,Prdt_15CoffeCrisp,6].OffsetPlace.Y=0
Ponto_STR[Pallet_2,Prdt_15CoffeCrisp,6].OffsetPlace.Z=0
Ponto_STR[Pallet_2,Prdt_15CoffeCrisp,6].OffsetPlace.A=0
Ponto_STR[Pallet_2,Prdt_15CoffeCrisp,6].OffsetPlace.B=0
Ponto_STR[Pallet_2,Prdt_15CoffeCrisp,6].OffsetPlace.C=0
;ENDFOLD
;ENDFOLD

;FOLD PLACE 7
;FOLD PROPRIEDADES
Ponto_STR[Pallet_2,Prdt_15CoffeCrisp,7].NumCaixas = 3
Ponto_STR[Pallet_2,Prdt_15CoffeCrisp,7].PickOp = 8
Ponto_STR[Pallet_2,Prdt_15CoffeCrisp,7].ConfGarraOp = 5
Ponto_STR[Pallet_2,Prdt_15CoffeCrisp,7].FechaGarraOp = 0
Ponto_STR[Pallet_2,Prdt_15CoffeCrisp,7].AbreGarraOp = 0
Ponto_STR[Pallet_2,Prdt_15CoffeCrisp,7].SensoresCaixa = 1234
Ponto_STR[Pallet_2,Prdt_15CoffeCrisp,7].TravaGarra = False
Ponto_STR[Pallet_2,Prdt_15CoffeCrisp,7].SkipGoHome = False
Ponto_STR[Pallet_2,Prdt_15CoffeCrisp,7].SkipSobeRelAtual = False
Ponto_STR[Pallet_2,Prdt_15CoffeCrisp,7].XApp1Place=P2_15CoffeCrisp_7_App1
Ponto_STR[Pallet_2,Prdt_15CoffeCrisp,7].XApp2Place=P2_15CoffeCrisp_7_App2
Ponto_STR[Pallet_2,Prdt_15CoffeCrisp,7].XPlace=P2_15CoffeCrisp_7_Place
;ENDFOLD
;FOLD OffsetPlace
Ponto_STR[Pallet_2,Prdt_15CoffeCrisp,7].OffsetPlace.X=0
Ponto_STR[Pallet_2,Prdt_15CoffeCrisp,7].OffsetPlace.Y=0
Ponto_STR[Pallet_2,Prdt_15CoffeCrisp,7].OffsetPlace.Z=0
Ponto_STR[Pallet_2,Prdt_15CoffeCrisp,7].OffsetPlace.A=0
Ponto_STR[Pallet_2,Prdt_15CoffeCrisp,7].OffsetPlace.B=0
Ponto_STR[Pallet_2,Prdt_15CoffeCrisp,7].OffsetPlace.C=0
;ENDFOLD
;ENDFOLD

;ENDFOLD
;FOLD LAYER 2: PLACE 8 ate 14
;FOLD PLACE 8
;FOLD PROPRIEDADES
Ponto_STR[Pallet_2,Prdt_15CoffeCrisp,8].NumCaixas = 1
Ponto_STR[Pallet_2,Prdt_15CoffeCrisp,8].PickOp = 6
Ponto_STR[Pallet_2,Prdt_15CoffeCrisp,8].ConfGarraOp = 5
Ponto_STR[Pallet_2,Prdt_15CoffeCrisp,8].FechaGarraOp = 0
Ponto_STR[Pallet_2,Prdt_15CoffeCrisp,8].AbreGarraOp = 0
Ponto_STR[Pallet_2,Prdt_15CoffeCrisp,8].SensoresCaixa = 1
Ponto_STR[Pallet_2,Prdt_15CoffeCrisp,8].TravaGarra = False
Ponto_STR[Pallet_2,Prdt_15CoffeCrisp,8].SkipGoHome = False
Ponto_STR[Pallet_2,Prdt_15CoffeCrisp,8].SkipSobeRelAtual = False
Ponto_STR[Pallet_2,Prdt_15CoffeCrisp,8].XApp1Place=P2_15CoffeCrisp_8_App1
Ponto_STR[Pallet_2,Prdt_15CoffeCrisp,8].XApp2Place=P2_15CoffeCrisp_8_App2
Ponto_STR[Pallet_2,Prdt_15CoffeCrisp,8].XPlace=P2_15CoffeCrisp_8_Place
;ENDFOLD
;FOLD OffsetPlace
Ponto_STR[Pallet_2,Prdt_15CoffeCrisp,8].OffsetPlace.X=0
Ponto_STR[Pallet_2,Prdt_15CoffeCrisp,8].OffsetPlace.Y=0
Ponto_STR[Pallet_2,Prdt_15CoffeCrisp,8].OffsetPlace.Z=0
Ponto_STR[Pallet_2,Prdt_15CoffeCrisp,8].OffsetPlace.A=0
Ponto_STR[Pallet_2,Prdt_15CoffeCrisp,8].OffsetPlace.B=0
Ponto_STR[Pallet_2,Prdt_15CoffeCrisp,8].OffsetPlace.C=0
;ENDFOLD
;ENDFOLD

;FOLD PLACE 9
;FOLD PROPRIEDADES
Ponto_STR[Pallet_2,Prdt_15CoffeCrisp,9].NumCaixas = 1
Ponto_STR[Pallet_2,Prdt_15CoffeCrisp,9].PickOp = 6
Ponto_STR[Pallet_2,Prdt_15CoffeCrisp,9].ConfGarraOp = 5
Ponto_STR[Pallet_2,Prdt_15CoffeCrisp,9].FechaGarraOp = 0
Ponto_STR[Pallet_2,Prdt_15CoffeCrisp,9].AbreGarraOp = 0
Ponto_STR[Pallet_2,Prdt_15CoffeCrisp,9].SensoresCaixa = 1
Ponto_STR[Pallet_2,Prdt_15CoffeCrisp,9].TravaGarra = False
Ponto_STR[Pallet_2,Prdt_15CoffeCrisp,9].SkipGoHome = False
Ponto_STR[Pallet_2,Prdt_15CoffeCrisp,9].SkipSobeRelAtual = False
Ponto_STR[Pallet_2,Prdt_15CoffeCrisp,9].XApp1Place=P2_15CoffeCrisp_9_App1
Ponto_STR[Pallet_2,Prdt_15CoffeCrisp,9].XApp2Place=P2_15CoffeCrisp_9_App2
Ponto_STR[Pallet_2,Prdt_15CoffeCrisp,9].XPlace=P2_15CoffeCrisp_9_Place
;ENDFOLD
;FOLD OffsetPlace
Ponto_STR[Pallet_2,Prdt_15CoffeCrisp,9].OffsetPlace.X=0
Ponto_STR[Pallet_2,Prdt_15CoffeCrisp,9].OffsetPlace.Y=0
Ponto_STR[Pallet_2,Prdt_15CoffeCrisp,9].OffsetPlace.Z=0
Ponto_STR[Pallet_2,Prdt_15CoffeCrisp,9].OffsetPlace.A=0
Ponto_STR[Pallet_2,Prdt_15CoffeCrisp,9].OffsetPlace.B=0
Ponto_STR[Pallet_2,Prdt_15CoffeCrisp,9].OffsetPlace.C=0
;ENDFOLD
;ENDFOLD

;FOLD PLACE 10
;FOLD PROPRIEDADES
Ponto_STR[Pallet_2,Prdt_15CoffeCrisp,10].NumCaixas = 1
Ponto_STR[Pallet_2,Prdt_15CoffeCrisp,10].PickOp = 6
Ponto_STR[Pallet_2,Prdt_15CoffeCrisp,10].ConfGarraOp = 5
Ponto_STR[Pallet_2,Prdt_15CoffeCrisp,10].FechaGarraOp = 0
Ponto_STR[Pallet_2,Prdt_15CoffeCrisp,10].AbreGarraOp = 0
Ponto_STR[Pallet_2,Prdt_15CoffeCrisp,10].SensoresCaixa = 1
Ponto_STR[Pallet_2,Prdt_15CoffeCrisp,10].TravaGarra = False
Ponto_STR[Pallet_2,Prdt_15CoffeCrisp,10].SkipGoHome = False
Ponto_STR[Pallet_2,Prdt_15CoffeCrisp,10].SkipSobeRelAtual = False
Ponto_STR[Pallet_2,Prdt_15CoffeCrisp,10].XApp1Place=P2_15CoffeCrisp_10_App1
Ponto_STR[Pallet_2,Prdt_15CoffeCrisp,10].XApp2Place=P2_15CoffeCrisp_10_App2
Ponto_STR[Pallet_2,Prdt_15CoffeCrisp,10].XPlace=P2_15CoffeCrisp_10_Place
;ENDFOLD
;FOLD OffsetPlace
Ponto_STR[Pallet_2,Prdt_15CoffeCrisp,10].OffsetPlace.X=0
Ponto_STR[Pallet_2,Prdt_15CoffeCrisp,10].OffsetPlace.Y=0
Ponto_STR[Pallet_2,Prdt_15CoffeCrisp,10].OffsetPlace.Z=0
Ponto_STR[Pallet_2,Prdt_15CoffeCrisp,10].OffsetPlace.A=0
Ponto_STR[Pallet_2,Prdt_15CoffeCrisp,10].OffsetPlace.B=0
Ponto_STR[Pallet_2,Prdt_15CoffeCrisp,10].OffsetPlace.C=0
;ENDFOLD
;ENDFOLD

;FOLD PLACE 11
;FOLD PROPRIEDADES
Ponto_STR[Pallet_2,Prdt_15CoffeCrisp,11].NumCaixas = 2
Ponto_STR[Pallet_2,Prdt_15CoffeCrisp,11].PickOp = 8
Ponto_STR[Pallet_2,Prdt_15CoffeCrisp,11].ConfGarraOp = 5
Ponto_STR[Pallet_2,Prdt_15CoffeCrisp,11].FechaGarraOp = 0
Ponto_STR[Pallet_2,Prdt_15CoffeCrisp,11].AbreGarraOp = 1
Ponto_STR[Pallet_2,Prdt_15CoffeCrisp,11].SensoresCaixa = 123
Ponto_STR[Pallet_2,Prdt_15CoffeCrisp,11].TravaGarra = True
Ponto_STR[Pallet_2,Prdt_15CoffeCrisp,11].SkipGoHome = False
Ponto_STR[Pallet_2,Prdt_15CoffeCrisp,11].SkipSobeRelAtual = False
Ponto_STR[Pallet_2,Prdt_15CoffeCrisp,11].XApp1Place=P2_15CoffeCrisp_11_App1
Ponto_STR[Pallet_2,Prdt_15CoffeCrisp,11].XApp2Place=P2_15CoffeCrisp_11_App2
Ponto_STR[Pallet_2,Prdt_15CoffeCrisp,11].XPlace=P2_15CoffeCrisp_11_Place
;ENDFOLD
;FOLD OffsetPlace
Ponto_STR[Pallet_2,Prdt_15CoffeCrisp,11].OffsetPlace.X=0
Ponto_STR[Pallet_2,Prdt_15CoffeCrisp,11].OffsetPlace.Y=0
Ponto_STR[Pallet_2,Prdt_15CoffeCrisp,11].OffsetPlace.Z=0
Ponto_STR[Pallet_2,Prdt_15CoffeCrisp,11].OffsetPlace.A=0
Ponto_STR[Pallet_2,Prdt_15CoffeCrisp,11].OffsetPlace.B=0
Ponto_STR[Pallet_2,Prdt_15CoffeCrisp,11].OffsetPlace.C=0
;ENDFOLD
;ENDFOLD

;FOLD PLACE 12
;FOLD PROPRIEDADES
Ponto_STR[Pallet_2,Prdt_15CoffeCrisp,12].NumCaixas = 2
Ponto_STR[Pallet_2,Prdt_15CoffeCrisp,12].PickOp = 8
Ponto_STR[Pallet_2,Prdt_15CoffeCrisp,12].ConfGarraOp = 5
Ponto_STR[Pallet_2,Prdt_15CoffeCrisp,12].FechaGarraOp = 0
Ponto_STR[Pallet_2,Prdt_15CoffeCrisp,12].AbreGarraOp = 1
Ponto_STR[Pallet_2,Prdt_15CoffeCrisp,12].SensoresCaixa = 123
Ponto_STR[Pallet_2,Prdt_15CoffeCrisp,12].TravaGarra = True
Ponto_STR[Pallet_2,Prdt_15CoffeCrisp,12].SkipGoHome = False
Ponto_STR[Pallet_2,Prdt_15CoffeCrisp,12].SkipSobeRelAtual = False
Ponto_STR[Pallet_2,Prdt_15CoffeCrisp,12].XApp1Place=P2_15CoffeCrisp_12_App1
Ponto_STR[Pallet_2,Prdt_15CoffeCrisp,12].XApp2Place=P2_15CoffeCrisp_12_App2
Ponto_STR[Pallet_2,Prdt_15CoffeCrisp,12].XPlace=P2_15CoffeCrisp_12_Place
;ENDFOLD
;FOLD OffsetPlace
Ponto_STR[Pallet_2,Prdt_15CoffeCrisp,12].OffsetPlace.X=0
Ponto_STR[Pallet_2,Prdt_15CoffeCrisp,12].OffsetPlace.Y=0
Ponto_STR[Pallet_2,Prdt_15CoffeCrisp,12].OffsetPlace.Z=0
Ponto_STR[Pallet_2,Prdt_15CoffeCrisp,12].OffsetPlace.A=0
Ponto_STR[Pallet_2,Prdt_15CoffeCrisp,12].OffsetPlace.B=0
Ponto_STR[Pallet_2,Prdt_15CoffeCrisp,12].OffsetPlace.C=0
;ENDFOLD
;ENDFOLD

;FOLD PLACE 13
;FOLD PROPRIEDADES
Ponto_STR[Pallet_2,Prdt_15CoffeCrisp,13].NumCaixas = 3
Ponto_STR[Pallet_2,Prdt_15CoffeCrisp,13].PickOp = 6
Ponto_STR[Pallet_2,Prdt_15CoffeCrisp,13].ConfGarraOp = 5
Ponto_STR[Pallet_2,Prdt_15CoffeCrisp,13].FechaGarraOp = 0
Ponto_STR[Pallet_2,Prdt_15CoffeCrisp,13].AbreGarraOp = 1
Ponto_STR[Pallet_2,Prdt_15CoffeCrisp,13].SensoresCaixa = 1234
Ponto_STR[Pallet_2,Prdt_15CoffeCrisp,13].TravaGarra = True
Ponto_STR[Pallet_2,Prdt_15CoffeCrisp,13].SkipGoHome = False
Ponto_STR[Pallet_2,Prdt_15CoffeCrisp,13].SkipSobeRelAtual = False
Ponto_STR[Pallet_2,Prdt_15CoffeCrisp,13].XApp1Place=P2_15CoffeCrisp_13_App1
Ponto_STR[Pallet_2,Prdt_15CoffeCrisp,13].XApp2Place=P2_15CoffeCrisp_13_App2
Ponto_STR[Pallet_2,Prdt_15CoffeCrisp,13].XPlace=P2_15CoffeCrisp_13_Place
;ENDFOLD
;FOLD OffsetPlace
Ponto_STR[Pallet_2,Prdt_15CoffeCrisp,13].OffsetPlace.X=0
Ponto_STR[Pallet_2,Prdt_15CoffeCrisp,13].OffsetPlace.Y=0
Ponto_STR[Pallet_2,Prdt_15CoffeCrisp,13].OffsetPlace.Z=0
Ponto_STR[Pallet_2,Prdt_15CoffeCrisp,13].OffsetPlace.A=0
Ponto_STR[Pallet_2,Prdt_15CoffeCrisp,13].OffsetPlace.B=0
Ponto_STR[Pallet_2,Prdt_15CoffeCrisp,13].OffsetPlace.C=0
;ENDFOLD
;ENDFOLD

;FOLD PLACE 14
;FOLD PROPRIEDADES
Ponto_STR[Pallet_2,Prdt_15CoffeCrisp,14].NumCaixas = 3
Ponto_STR[Pallet_2,Prdt_15CoffeCrisp,14].PickOp = 6
Ponto_STR[Pallet_2,Prdt_15CoffeCrisp,14].ConfGarraOp = 5
Ponto_STR[Pallet_2,Prdt_15CoffeCrisp,14].FechaGarraOp = 0
Ponto_STR[Pallet_2,Prdt_15CoffeCrisp,14].AbreGarraOp = 1
Ponto_STR[Pallet_2,Prdt_15CoffeCrisp,14].SensoresCaixa = 1234
Ponto_STR[Pallet_2,Prdt_15CoffeCrisp,14].TravaGarra = True
Ponto_STR[Pallet_2,Prdt_15CoffeCrisp,14].SkipGoHome = False
Ponto_STR[Pallet_2,Prdt_15CoffeCrisp,14].SkipSobeRelAtual = False
Ponto_STR[Pallet_2,Prdt_15CoffeCrisp,14].XApp1Place=P2_15CoffeCrisp_14_App1
Ponto_STR[Pallet_2,Prdt_15CoffeCrisp,14].XApp2Place=P2_15CoffeCrisp_14_App2
Ponto_STR[Pallet_2,Prdt_15CoffeCrisp,14].XPlace=P2_15CoffeCrisp_14_Place
;ENDFOLD
;FOLD OffsetPlace
Ponto_STR[Pallet_2,Prdt_15CoffeCrisp,14].OffsetPlace.X=0
Ponto_STR[Pallet_2,Prdt_15CoffeCrisp,14].OffsetPlace.Y=0
Ponto_STR[Pallet_2,Prdt_15CoffeCrisp,14].OffsetPlace.Z=0
Ponto_STR[Pallet_2,Prdt_15CoffeCrisp,14].OffsetPlace.A=0
Ponto_STR[Pallet_2,Prdt_15CoffeCrisp,14].OffsetPlace.B=0
Ponto_STR[Pallet_2,Prdt_15CoffeCrisp,14].OffsetPlace.C=0
;ENDFOLD
;ENDFOLD

;ENDFOLD
;ENDFOLD

;ENDFOLD
END
